(* test hex_to_dword *)
good := good AND HEX_TO_DWORD('0ff') = 255;
good := good AND HEX_TO_DWORD('00') = 0;
good := good AND HEX_TO_DWORD('1') = 1;
good := good AND HEX_TO_DWORD('0A') = 10;
good := good AND HEX_TO_DWORD('0F') = 15;
good := good AND HEX_TO_DWORD('0a') = 10;
good := good AND HEX_TO_DWORD('0f') = 15;
good := good AND HEX_TO_DWORD('00009') = 9;

(* test lowercase *)
good := good AND LOWERCASE('FGTHZuz2345KJGH') = 'fgthzuz2345kjgh';

(* test mirror *)
good := good AND MIRROR('123456789 abc') = 'cba 987654321';

(* test real_to_strf *)
good := good AND REAL_TO_STRF(pi1,2) = '3.14';
good := good AND REAL_TO_STRF(0.015,2) = '0.02';
good := good AND REAL_TO_STRF(0.015,4) = '0.0150';
good := good AND REAL_TO_STRF(0.015,0) = '0';
good := good AND REAL_TO_STRF(3.015,1) = '3.0';
good := good AND REAL_TO_STRF(1234.49967,0) = '1234';
good := good AND REAL_TO_STRF(1234.49967,1) = '1234.5';
good := good AND REAL_TO_STRF(1234.49967,2) = '1234.50';
good := good AND REAL_TO_STRF(1234.49964,3) = '1234.500';
good := good AND REAL_TO_STRF(14.49967,4) = '14.4997';
good := good AND REAL_TO_STRF(1.49967,5) = '1.49967';
good := good AND REAL_TO_STRF(1.49967,6) = '1.499670';

(* test replace_all *)
good := good AND REPLACE_ALL('ab12cd12ef12gh','12','') = 'abcdefgh';
good := good AND REPLACE_ALL('ab12cd12ef12gh','12','21') = 'ab21cd21ef21gh';
good := good AND REPLACE_ALL('ab12cd12ef12gh','12','12') = 'ab12cd12ef12gh';

(* test trim *)
good := good AND TRIM(' ab  cd ef  gh ') = 'abcdefgh';


(* test trim1 *)
good := good AND TRIM1(' ab  cd ef  gh ') = 'ab cd ef gh';

(* test uppercase *)
good := good AND UPPERCASE('fgTHZu z2345KJGH') = 'FGTHZU Z2345KJGH';

(* test capitalize *)
good := good AND CAPITALIZE('hugo wallenstein 123') = 'Hugo Wallenstein 123';

(* test to_upper and to lower *)
FOR t := 0 TO 255 DO
	i := INT_TO_BYTE(t);
	CASE i OF
	0..64:
		good := good AND TO_LOWER(i) = i AND TO_UPPER(i) = i;
	65..90: (* uppercase letters *)
		good := good AND TO_UPPER(i) = i;
		good := good AND TO_LOWER(i) = i + 32;
	91..96:
		good := good AND TO_LOWER(i) = i AND TO_UPPER(i) = i;
	97..122: (* small letters *)
		good := good AND TO_UPPER(i) = i - 32;
		good := good AND TO_LOWER(i) = i;
	123..191:
		good := good AND TO_LOWER(i) = i AND TO_UPPER(i) = i;
	192..214: (* extended uppercase letters *)
		good := good AND TO_UPPER(i) = i;
		good := good AND TO_LOWER(i) = i + 32;
	215:
		good := good AND TO_LOWER(i) = i AND TO_UPPER(i) = i;
	216..222: (* extended uppercase letters *)
		good := good AND TO_UPPER(i) = i;
		good := good AND TO_LOWER(i) = i + 32;
	223:
		good := good AND TO_LOWER(i) = i AND TO_UPPER(i) = i;
	224..246: (* extended lowercase letters *)
		good := good AND TO_UPPER(i) = i-32;
		good := good AND TO_LOWER(i) = i;
	247:
		good := good AND TO_LOWER(i) = i AND TO_UPPER(i) = i;
	248..254: (* extended lowercase letters *)
		good := good AND TO_UPPER(i) = i-32;
		good := good AND TO_LOWER(i) = i;
	255:
		good := good AND TO_LOWER(i) = i AND TO_UPPER(i) = i;
	END_CASE;
	temp := CONCAT(INT_TO_STRING(t),' > ');
	temp := CONCAT(temp,CHR(TO_UPPER(i)));
	temp := CONCAT(temp,' > ');
	temp := CONCAT(temp,CHR(TO_LOWER(i)));
END_FOR;

(* test isc funktionen *)
FOR t := 0 TO 255 DO
	i := INT_TO_BYTE(t);
	CASE i OF
	0..31:
		good := good AND ISC_CTRL(i) = TRUE;
		good := good AND ISC_NUM(i) = FALSE;
		good := good AND ISC_ALPHA(i) = FALSE;
		good := good AND ISC_HEX(i) = FALSE;
		good := good AND ISC_LOWER(i) = FALSE;
		good := good AND ISC_UPPER(i) = FALSE;
	32..47:
		good := good AND ISC_CTRL(i) = FALSE;
		good := good AND ISC_NUM(i) = FALSE;
		good := good AND ISC_ALPHA(i) = FALSE;
		good := good AND ISC_HEX(i) = FALSE;
		good := good AND ISC_LOWER(i) = FALSE;
		good := good AND ISC_UPPER(i) = FALSE;
	48..57:
		good := good AND ISC_CTRL(i) = FALSE;
		good := good AND ISC_NUM(i) = TRUE;
		good := good AND ISC_ALPHA(i) = FALSE;
		good := good AND ISC_HEX(i) = TRUE;
		good := good AND ISC_LOWER(i) = FALSE;
		good := good AND ISC_UPPER(i) = FALSE;
	58..64:
		good := good AND ISC_CTRL(i) = FALSE;
		good := good AND ISC_NUM(i) = FALSE;
		good := good AND ISC_ALPHA(i) = FALSE;
		good := good AND ISC_HEX(i) = FALSE;
		good := good AND ISC_LOWER(i) = FALSE;
		good := good AND ISC_UPPER(i) = FALSE;
	65..70:
		good := good AND ISC_CTRL(i) = FALSE;
		good := good AND ISC_NUM(i) = FALSE;
		good := good AND ISC_ALPHA(i) = TRUE;
		good := good AND ISC_HEX(i) = TRUE;
		good := good AND ISC_LOWER(i) = FALSE;
		good := good AND ISC_UPPER(i) = TRUE;
	75..90:
		good := good AND ISC_CTRL(i) = FALSE;
		good := good AND ISC_NUM(i) = FALSE;
		good := good AND ISC_ALPHA(i) = TRUE;
		good := good AND ISC_HEX(i) = FALSE;
		good := good AND ISC_LOWER(i) = FALSE;
		good := good AND ISC_UPPER(i) = TRUE;
	91..96:
		good := good AND ISC_CTRL(i) = FALSE;
		good := good AND ISC_NUM(i) = FALSE;
		good := good AND ISC_ALPHA(i) = FALSE;
		good := good AND ISC_HEX(i) = FALSE;
		good := good AND ISC_LOWER(i) = FALSE;
		good := good AND ISC_UPPER(i) = FALSE;
	97..102:
		good := good AND ISC_CTRL(i) = FALSE;
		good := good AND ISC_NUM(i) = FALSE;
		good := good AND ISC_ALPHA(i) = TRUE;
		good := good AND ISC_HEX(i) = TRUE;
		good := good AND ISC_LOWER(i) = TRUE;
		good := good AND ISC_UPPER(i) = FALSE;
	103..122:
		good := good AND ISC_CTRL(i) = FALSE;
		good := good AND ISC_NUM(i) = FALSE;
		good := good AND ISC_ALPHA(i) = TRUE;
		good := good AND ISC_HEX(i) = FALSE;
		good := good AND ISC_LOWER(i) = TRUE;
		good := good AND ISC_UPPER(i) = FALSE;
	123..126:
		good := good AND ISC_CTRL(i) = FALSE;
		good := good AND ISC_NUM(i) = FALSE;
		good := good AND ISC_ALPHA(i) = FALSE;
		good := good AND ISC_HEX(i) = FALSE;
		good := good AND ISC_LOWER(i) = FALSE;
		good := good AND ISC_UPPER(i) = FALSE;
	127:
		good := good AND ISC_CTRL(i) = TRUE;
		good := good AND ISC_NUM(i) = FALSE;
		good := good AND ISC_ALPHA(i) = FALSE;
		good := good AND ISC_HEX(i) = FALSE;
		good := good AND ISC_LOWER(i) = FALSE;
		good := good AND ISC_UPPER(i) = FALSE;
	128..191:
		good := good AND ISC_CTRL(i) = FALSE;
		good := good AND ISC_NUM(i) = FALSE;
		good := good AND ISC_ALPHA(i) = FALSE;
		good := good AND ISC_HEX(i) = FALSE;
		good := good AND ISC_LOWER(i) = FALSE;
		good := good AND ISC_UPPER(i) = FALSE;
	192..214:
		good := good AND ISC_CTRL(i) = FALSE;
		good := good AND ISC_NUM(i) = FALSE;
		good := good AND ISC_ALPHA(i) = EXTENDED_ASCII;
		good := good AND ISC_HEX(i) = FALSE;
		good := good AND ISC_LOWER(i) = FALSE;
		good := good AND ISC_UPPER(i) = EXTENDED_ASCII;
	215:
		good := good AND ISC_CTRL(i) = FALSE;
		good := good AND ISC_NUM(i) = FALSE;
		good := good AND ISC_ALPHA(i) = FALSE;
		good := good AND ISC_HEX(i) = FALSE;
		good := good AND ISC_LOWER(i) = FALSE;
		good := good AND ISC_UPPER(i) = FALSE;
	216..222:
		good := good AND ISC_CTRL(i) = FALSE;
		good := good AND ISC_NUM(i) = FALSE;
		good := good AND ISC_ALPHA(i) = EXTENDED_ASCII;
		good := good AND ISC_HEX(i) = FALSE;
		good := good AND ISC_LOWER(i) = FALSE;
		good := good AND ISC_UPPER(i) = EXTENDED_ASCII;
	223:
		good := good AND ISC_CTRL(i) = FALSE;
		good := good AND ISC_NUM(i) = FALSE;
		good := good AND ISC_ALPHA(i) = TRUE;
		good := good AND ISC_HEX(i) = FALSE;
		good := good AND ISC_LOWER(i) = TRUE;
		good := good AND ISC_UPPER(i) = FALSE;
	224..246:
		good := good AND ISC_CTRL(i) = FALSE;
		good := good AND ISC_NUM(i) = FALSE;
		good := good AND ISC_ALPHA(i) = EXTENDED_ASCII;
		good := good AND ISC_HEX(i) = FALSE;
		good := good AND ISC_LOWER(i) = EXTENDED_ASCII;
		good := good AND ISC_UPPER(i) = FALSE;
	247:
		good := good AND ISC_CTRL(i) = FALSE;
		good := good AND ISC_NUM(i) = FALSE;
		good := good AND ISC_ALPHA(i) = FALSE;
		good := good AND ISC_HEX(i) = FALSE;
		good := good AND ISC_LOWER(i) = FALSE;
		good := good AND ISC_UPPER(i) = FALSE;
	248..254:
		good := good AND ISC_CTRL(i) = FALSE;
		good := good AND ISC_NUM(i) = FALSE;
		good := good AND ISC_ALPHA(i) = EXTENDED_ASCII;
		good := good AND ISC_HEX(i) = FALSE;
		good := good AND ISC_LOWER(i) = EXTENDED_ASCII;
		good := good AND ISC_UPPER(i) = FALSE;
	255:
		good := good AND ISC_CTRL(i) = FALSE;
		good := good AND ISC_NUM(i) = FALSE;
		good := good AND ISC_ALPHA(i) = TRUE;
		good := good AND ISC_HEX(i) = FALSE;
		good := good AND ISC_LOWER(i) = TRUE;
		good := good AND ISC_UPPER(i) = FALSE;
	END_CASE;
END_FOR;

(* code test *)
FOR t := 1 TO 255 DO
	good := good AND CODE(CHR(INT_TO_BYTE(t)),1) = INT_TO_BYTE(t);
END_FOR;
temp := '0123456789';
good := good AND CODE(temp,1) = 48;
good := good AND CODE(temp,0) = 0;
good := good AND CODE(temp,11) = 0;
good := good AND CODE(temp,10) = 57;

(* test is_cc is_ncc*)
good := good AND IS_CC('0123456789','0123456789') = TRUE;
good := good AND IS_CC('0 123456789','0123456789') = FALSE;
good := good AND IS_CC('','+-abcdefgh ') = FALSE;
good := good AND IS_NCC('0123456789','+-abcdefgh ') = TRUE;
good := good AND IS_NCC('+0123456789','+-abcdefgh ') = FALSE;
good := good AND IS_NCC('','+-abcdefgh ') = TRUE;

(* test trime *)
good := good AND TRIME('') = '';
good := good AND TRIME('this one') = 'this one';
good := good AND TRIME('  that one   ') = 'that one';

(* test fill *)
good := good AND FILL(32,3) = '   ';
good := good AND FILL(32,0) = '';

(* test fix *)
good := good AND FIX('that one',3,32,0) = 'tha';
good := good AND FIX('this',7,32,0) = 'this   ';
good := good AND FIX('',3,32,0) = '   ';
good := good AND FIX('that one',0,32,0) = '';
good := good AND FIX('that one',3,32,1) = 'one';
good := good AND FIX('this',7,32,1) = '   this';
good := good AND FIX('',3,32,1) = '   ';
good := good AND FIX('that one',0,32,1) = '';
good := good AND FIX('that one',3,32,2) = 'tha';
good := good AND FIX('this',7,32,2) = ' this  ';
good := good AND FIX('',3,32,2) = '   ';
good := good AND FIX('that one',0,32,2) = '';

(* test charcode and charname *)
FOR i := 0 TO 40 DO
	s1 := CHARNAME(i);
	good := good AND (CHARCODE(s1) = i);
END_FOR
good := good AND (CHARNAME(128) = 'euro');
good := good AND (CHARCODE('euro') = 128);




(* revision history
hm	26. mar. 2008	rev 1.0
	original release

hm	29. mar. 2008	rev 1.1
	added trime, fix and fill

hm	29. mar. 2008	rev 1.2
	changed parameter in test fix for new version of fix
	more test for dword_strH

hm	30. mar. 2008	rev 1.3
	added further test for replace UML with € sign

hm	18. may 2008	rev 1.4
	added tests for charcode and charname

*)
END_FUNCTION_BLOCK

(* POU String/FIND_CHAR, ST *)
FUNCTION FIND_CHAR : INT
VAR_INPUT
	str : STRING(STRING_LENGTH);
	pos : INT;
END_VAR
VAR
	i: INT;
	pt : POINTER TO ARRAY[1..255] OF BYTE;
	stop: INT;
	X: BYTE;
END_VAR

(*
version 1.2	29. mar. 2008
programmer 	hugo
tested by		tobias

find_char searches str and returns the starting position of the first character that is not a control character.
control characters are the ascii character 00 .. 31 and 127

*)
pt := ADR(str);
stop := LEN(str);
FOR i := MAX(pos,1) TO stop DO;
	X := pt^[i];
	IF (extended_ascii AND X > 31 AND X <> 127) OR (NOT extended_ascii AND X > 31 AND X < 127) THEN
		FIND_CHAR := i;
		RETURN;
	END_IF;
END_FOR;
FIND_CHAR := 0;


(* revision history
hm	29. feb 2008	rev 1.0
	original version

hm	26. mar. 2008	rev 1.1
	char will now accept extended ascii

hm	29. mar. 2008	rev 1.2
	changed STRING to STRING(STRING_LENGTH)
*)
END_FUNCTION

(* POU String/IS_ALNUM, ST *)
FUNCTION IS_ALNUM : BOOL
VAR_INPUT
	str : STRING(STRING_LENGTH);
END_VAR
VAR
	L: INT;
	pt : POINTER TO BYTE;
	pos: INT;
END_VAR

(*
version 1.1	29. mar. 2008
programmer 		kurt
tested by		hugo

ISC_ALNUM testet ob in einem string nur Zahlen 0..9 vorkommen.

*)
PT := ADR(str);
L := LEN(str);
FOR pos := 1 TO L DO
	IF NOT (ISC_ALPHA(pt^) OR ISC_NUM(pt^)) THEN
		IS_ALNUM := FALSE;
		RETURN;
	END_IF;
    	PT := PT + 1;
END_FOR;
IS_ALNUM := L > 0;


(* revision history
hm	29. feb 2008	rev 1.0
	original version

hm	29. mar. 2008	rev 1.1
	changed STRING to STRING(STRING_LENGTH)
*)
END_FUNCTION

(* POU String/ISC_ALPHA, ST *)
FUNCTION ISC_ALPHA : BOOL
VAR_INPUT
	IN : BYTE;
END_VAR
VAR
END_VAR

(*
version 1.0	6. mar 2008
programmer 	oscat
tested by		hugo

ISC_ALPHA checks if a character is a..z or A..Z.

*)
IF extended_ascii THEN
	ISC_ALPHA := (in > 64 AND in < 91) OR (in > 191  AND in <> 215 AND in <> 247) OR (in > 96 AND in < 123);
ELSE
	ISC_ALPHA := (IN > 64 AND IN < 91) OR (in > 96 AND in < 123);
END_IF;

(* revision history
hm		6. mar. 2008	rev 1.0
	original version

*)
END_FUNCTION

(* POU String/ISC_NUM, ST *)
FUNCTION ISC_NUM : BOOL
VAR_INPUT
	IN : BYTE;
END_VAR
VAR
END_VAR

(*
version 1.0	6. mar 2008
programmer 	oscat
tested by		hugo

ISC_NUM checks if a character is 0..9.

*)
ISC_NUM := IN > 47 AND IN < 58;

(* revision history
hm		6. mar. 2008	rev 1.0
	original version

*)
END_FUNCTION

(* POU String/CHR, ST *)
FUNCTION CHR : STRING(1)
VAR_INPUT
	C : BYTE;
END_VAR
VAR
	PT : POINTER TO BYTE;
END_VAR

(*
version 1.2	29. mar. 2008
programmer 	hugo
tested by		tobias

CHR creates a character from a byte input and stuffs it in a one character length string.

*)
PT := ADR(CHR);
PT^ := C;
pt := pt + 1;
pt^ := 0;

(* revision history
hm	16 jan 2007		rev 1.0
	original version

hm	4. feb. 2008	rev 1.1
	return string would not be terminated properly

hm	29. mar. 2008	rev 1.2
	changed STRING to STRING(1)
*)
END_FUNCTION

(* POU String/IS_ALPHA, ST *)
FUNCTION IS_ALPHA : BOOL
VAR_INPUT
	str : STRING(STRING_LENGTH);
END_VAR
VAR
	L: INT;
	pt : POINTER TO BYTE;
	pos: INT;
END_VAR

(*
version 1.1	29. mar. 2008
programmer 		kurt
tested by		hugo

IS_ALPHA testet ob in einem string nur Zeichen a-z oder A - Z vorkommen.

*)
PT := ADR(str);
L := LEN(str);
FOR pos := 1 TO L DO
	IF NOT ISC_ALPHA(pt^) THEN
		IS_ALPHA := FALSE;
		RETURN;
	END_IF;
    	PT := PT + 1;
END_FOR;
IS_ALPHA := L > 0;


(* revision history
hm	29. feb 2008	rev 1.0
	original version

hm	29. mar. 2008	rev 1.1
	changed STRING to STRING(STRING_LENGTH)
*)
END_FUNCTION

(* POU String/IS_CTRL, ST *)
FUNCTION IS_CTRL : BOOL
VAR_INPUT
	str : STRING(STRING_LENGTH);
END_VAR
VAR
	L: INT;
	pt : POINTER TO BYTE;
	pos: INT;
END_VAR

(*
version 1.1	29. mar 2008
programmer 		kurt
tested by		hugo

IS_CTRL testet ob in einem string nur Steuerzeichen (Char < 32) vorkommen.

*)
PT := ADR(str);
L := LEN(str);
FOR pos := 1 TO L DO
	IF NOT (ISC_CTRL(pt^)) THEN
		IS_CTRL := FALSE;
		RETURN;
	END_IF;
    	PT := PT + 1;
END_FOR;
IS_CTRL := L > 0;


(* revision history
hm	29. feb. 2008	rev 1.0
	original version

hm	29. mar. 2008	rev 1.1
	changed STRING to STRING(STRING_LENGTH)
*)
END_FUNCTION

(* POU String/ISC_CTRL, ST *)
FUNCTION ISC_CTRL : BOOL
VAR_INPUT
	IN : BYTE;
END_VAR
VAR
END_VAR

(*
version 1.0	6. mar 2008
programmer 	oscat
tested by		hugo

ISC_ALPHA checks if a character is a control character.

*)
ISC_CTRL := IN < 32 OR IN = 127;

(* revision history
hm		6. mar. 2008	rev 1.0
	original version

*)
END_FUNCTION

(* POU String/IS_HEX, ST *)
FUNCTION IS_HEX : BOOL
VAR_INPUT
	str : STRING(STRING_LENGTH);
END_VAR
VAR
	L: INT;
	pt : POINTER TO BYTE;
	pos: INT;
END_VAR

(*
version 1.1	29. mar. 2008
programmer 		kurt
tested by		hugo

IS_HEX testet ob in einem string nur Zahlen 0..9 oder A..F oder a..f  vorkommen.

*)
PT := ADR(str);
L := LEN(str);
FOR pos := 1 TO L DO
	IF NOT (ISC_HEX(pt^)) THEN
		IS_HEX := FALSE;
		RETURN;
	END_IF;
    	PT := PT + 1;
END_FOR;
IS_HEX := L > 0;


(* revision history
hm	29. feb 2008	rev 1.0
	original version

hm	29. mar. 2008	rev 1.1
	changed STRING to STRING(STRING_LENGTH)
*)
END_FUNCTION

(* POU String/ISC_HEX, ST *)
FUNCTION ISC_HEX : BOOL
VAR_INPUT
	IN : BYTE;
END_VAR
VAR
END_VAR

(*
version 1.0	6. mar 2008
programmer 	oscat
tested by		hugo

ISC_HEX checks if a character is 0..9, A..F, a..f.

*)
ISC_HEX := (IN > 47 AND IN < 58) OR (IN > 64 AND IN < 71) OR (IN > 96 AND IN < 103);

(* revision history
hm		6. mar. 2008	rev 1.0
	original version

*)
END_FUNCTION

(* POU String/IS_LOWER, ST *)
FUNCTION IS_LOWER : BOOL
VAR_INPUT
	str : STRING(STRING_LENGTH);
END_VAR
VAR
	l: INT;
	pt : POINTER TO BYTE;
	pos: INT;
END_VAR

(*
version 1.1	29. mar. 2008
programmer 		kurt
tested by		hugo

IS_LOWER testet ob in einem string nur kleinbuchstaben vorkommen.

*)
PT := ADR(str);
L := LEN(str);
FOR pos := 1 TO L DO
	IF NOT (ISC_LOWER(pt^)) THEN
		IS_LOWER := FALSE;
		RETURN;
	END_IF;
    	PT := PT + 1;
END_FOR;
IS_LOWER := L > 0;


(* revision history
hm	29. feb 2008	rev 1.0
	original version

hm	29. mar. 2008	rev 1.1
	changed STRING to STRING(STRING_LENGTH)
*)
END_FUNCTION

(* POU String/ISC_LOWER, ST *)
FUNCTION ISC_LOWER : BOOL
VAR_INPUT
	IN : BYTE;
END_VAR
VAR
END_VAR

(*
version 1.0	6 mar 2008
programmer 	hugo
tested by		tobias

isc_lower checks if a character is lowercase.

*)
IF extended_ascii THEN
	ISC_LOWER := ((in > 96) AND (in < 123)) OR ((in > 222) AND (in <> 247));
ELSE
	ISC_LOWER := ((in > 96) AND (in < 123));
END_IF;

(* revision history
hm		6. mar 2008	rev 1.0
	original version

*)
END_FUNCTION

(* POU String/IS_UPPER, ST *)
FUNCTION IS_UPPER : BOOL
VAR_INPUT
	str : STRING(STRING_LENGTH);
END_VAR
VAR
	L: INT;
	pt : POINTER TO BYTE;
	pos: INT;
END_VAR

(*
version 1.1	29. mar. 2008
programmer 		kurt
tested by		hugo

IS_UPPER testet ob in einem string keine Kleinbuchstaben vorkommen.

*)
PT := ADR(str);
L := LEN(str);
FOR pos := 1 TO L DO
	IF NOT (ISC_UPPER(pt^)) THEN
		IS_UPPER := FALSE;
		RETURN;
	END_IF;
    	PT := PT + 1;
END_FOR;
IS_UPPER := L > 0;


(* revision history
hm	29. feb 2008	rev 1.0
	original version

hm	29. mar. 2008	rev 1.1
	changed STRING to STRING(STRING_LENGTH)
*)
END_FUNCTION

(* POU String/ISC_UPPER, ST *)
FUNCTION ISC_UPPER : BOOL
VAR_INPUT
	IN : BYTE;
END_VAR
VAR
END_VAR

(*
version 1.0	6 mar 2008
programmer 	hugo
tested by		tobias

ISC_upper checks if a character is uppercase

*)
IF extended_ascii THEN
	ISC_UPPER :=  ((in > 64) AND (in < 91)) OR (((in > 191) AND (in < 223)) AND (in <> 215));
ELSE
	ISC_UPPER := ((in > 64) AND (in < 91));
END_IF;


(* revision history
hm		6. mar 2008	rev 1.0
	original version

*)
END_FUNCTION

(* POU String/IS_NUM, ST *)
FUNCTION IS_NUM : BOOL
VAR_INPUT
	str : STRING(STRING_LENGTH);
END_VAR
VAR
	L : INT;
	pt : POINTER TO BYTE;
	pos: INT;
END_VAR

(*
version 1.1	29. mar. 2008
programmer 		kurt
tested by		hugo

IS_NUM testet ob in einem string nur Zahlen 0..9 vorkommen.

*)
PT := ADR(str);
L := LEN(str);
FOR pos := 1 TO L DO
	IF NOT (ISC_NUM(pt^)) THEN
		IS_NUM := FALSE;
		RETURN;
	END_IF;
    	PT := PT + 1;
END_FOR;
IS_NUM := L > 0;


(* revision history
hm	29. feb 2008	rev 1.0
	original version

hm	29. mar. 2008	rev 1.1
	changed STRING to STRING(STRING_LENGTH)
*)
END_FUNCTION

(* POU String/REPLACE_UML, ST *)
FUNCTION REPLACE_UML : STRING(STRING_LENGTH)
VAR_INPUT
	str : STRING(STRING_LENGTH);
END_VAR
VAR
	L : INT;
	pt : POINTER TO BYTE;
	pto : POINTER TO BYTE;
	ptm : POINTER TO BYTE;
	pt1, pt2 : POINTER TO BYTE;
	su : STRING(2);
	pos : INT;
END_VAR

(*
version 1.1	29. mar. 2008
programmer 		kurt
tested by		hugo

REPLACE_UML replaces all occurences of Ä,Ö,Ü and ä,ö,ü,ß with Ae, ae, Oe, oe, Ue, ue and ss.

*)
PT := ADR(str);
pto := ADR(REPLACE_UML);
ptm := pto + INT_TO_DWORD(string_length);
pt1 := ADR(su);
pt2 := pt1 + 1;
L := LEN(str);
WHILE pos < L AND pos < string_length DO
	IF pt^ < 127 THEN
		(* no uml character simlply copy the character*)
		pto^ := pt^;
	ELSE
		(* convert the uml character *)
		su := TO_UML(pt^);
		(* we must make sure pointer are not out of range *)
		pto^ := pt1^;
		IF pto < ptm AND pt2^ > 0 THEN
			pto := pto + 1;
			pto^ := pt2^;
		END_IF;
	END_IF;
	(* increment pointers *)
	pt := pt + 1;
	pto := pto + 1;
	pos := pos + 1;
END_WHILE;

(* properly close the output string *)
pto^ := 0;


(* revision history
hm	29. feb 2008	rev 1.0
	original version

hm	29. mar. 2008	rev 1.1
	changed STRING to STRING(STRING_LENGTH)
	new code to avoid pointer out of range
	use new function to_uml
*)
END_FUNCTION

(* POU String/TO_UML, ST *)
FUNCTION TO_UML : STRING(2)
VAR_INPUT
	IN : BYTE;
END_VAR
VAR
END_VAR

(*
version 1.0	29. mar. 2008
programmer 		hugo
tested by		tobias

to_uml converts a character above 127 to a two digit character below 127.
the character Ä is converted to Ae

*)
CASE in OF
	196:	(* Ä *)
		TO_UML := 'Ae';
	214:	(* Ö *)
		TO_UML := 'Oe';
	220:	(* Ü *)
		TO_UML := 'Ue';
	223:	(* ß *)
		TO_UML := 'ss';
	228:	(* ä *)
		TO_UML := 'ae';
	246:	(* ö *)
		TO_UML := 'oe';
	252:	(* ü *)
		TO_UML := 'ue';
ELSE
	TO_UML := CHR(IN);
END_CASE;



(* revision history
hm	29. mar. 2008	rev 1.0
	original version

*)
END_FUNCTION

(* POU String/BYTE_TO_STRH, ST *)
FUNCTION BYTE_TO_STRH : STRING(2)
VAR_INPUT
	IN : BYTE;
END_VAR
VAR
	temp : BYTE;
	PT : POINTER TO BYTE;
END_VAR

(*
version 1.3	29 mar. 2008
programmer 	hugo
tested by		tobias

BYTE_TO_STRINGH converts a Byte to a String of Hexadecimal represented by '0' .. '9' and 'A' .. 'F'.
The lowest order Character will be on the right and the high order Character on the left.

*)
(* read pointer to output string *)
PT := ADR(BYTE_TO_STRH);
(* calculate high order hex value *)
temp := SHR(in,4);
(* convert value to hex character *)
IF temp <= 9 THEN temp := temp + 48; ELSE temp := temp + 55; END_IF;
(* write friat character to output string *)
PT^ := temp;
(* calculate low order hex value *)
temp := in AND 2#00001111;
IF temp <= 9 THEN temp := temp + 48; ELSE temp := temp + 55; END_IF;
(* increment pointer and wirte low order character *)
pt := pt + 1;
pt^ := temp;
(* set pointer at the end of the output string and close the string with 0 *)
pt := pt + 1;
pt^:= 0;


(* code before rev 1.2
FOR i := 1 TO 2 DO
	X := in AND 2#1111;
	IF X <= 9 THEN X := X + 48; ELSE X := X + 55; END_IF;
	Cx := CHR(X);
	temp := CONCAT(Cx, temp);
	in := SHR(in,4);
END_FOR;
BYTE_TO_STRH := temp;
*)

(* revision history

hm	9.6.2007		rev 1.0		
	original version 

hm	11.9.2007		rev 1.1		
	changed coding for compatibility with twincat, under twincat concat cannot have a function as argument.	

hm	15 dec 2007		REV 1.2
	changed code for higher performance

hm	29. mar. 2008	rev 1.3
	changed STRING to STRING(2)
*)
END_FUNCTION

(* POU String/DWORD_TO_STRF, ST *)
FUNCTION DWORD_TO_STRF : STRING(20)
VAR_INPUT
	IN : DWORD;
	N : INT;
END_VAR
VAR
END_VAR

(*
version 1.0	26 jan 2007
programmer 	hugo
tested by		tobias

dword_to_strF converts a DWORD, BYTE or Word to a fixed length String.
the string will be filled with leading zeroes to achieve the fixed length, or if too long, the lowest digits will be used.
the maximum allowed length is 20 mdigits.

for example:	dword_to_strf(123,4) = '0123' 
				dword_to_strf(123,2) = '23'
*)
(* limit N to max 20 characters *)
(* convert dword to string first and cut to length N *)
DWORD_TO_STRF := FIX(DWORD_TO_STRING(in),LIMIT(0,N,20),48,1);


(* revision history
hm	26. jan.2007	rev 1.0		
	original version

hm	29. mar. 2008	rev 1.1
	changed STRING to STRING(20)
	limit the output string to max 20 digits
*)
END_FUNCTION

(* POU String/FIX, ST *)
FUNCTION FIX : STRING(STRING_LENGTH)
VAR_INPUT
	str : STRING(STRING_LENGTH);
	L : INT;
	C : BYTE;
	M : INT;
END_VAR
VAR
	N : INT;
	SX: STRING(STRING_LENGTH);
END_VAR

(*
version 1.0	29. mar. 2008
programmer 	hugo
tested by	tobias

the function fix truncates a string at length L 
or if the string is shorter then L it will be filled with ending Spaces till its length = N.

*)
(* make sure L does not exceed the limits of a string *)
N := LIMIT(0,L,STRING_LENGTH) - LEN(str);
IF N <= 0 THEN
	(* truncate the string at length N *)
	IF M = 1 THEN
		FIX := RIGHT(str,L);
	ELSE
		FIX := LEFT(str,L);
	END_IF;
ELSIF M = 1 THEN
	(* connect fill characters at the beginning *)
	sx := FILL(C,N);
	FIX := CONCAT(sx,str);
ELSIF M = 2 THEN
	(* center str beween fill characters *)
	(* for an uneven number of fill characters, there is one more at the end *)
	sx := FILL(C,SHR(N+1,1));
	FIX := CONCAT(str,sx);
	SX := LEFT(sx,SHR(N,1));
	FIX := CONCAT(sx,FIX);
ELSE
	(* connect fill characters at the end *)
	SX := FILL(C,N);
	FIX := CONCAT(str,SX);
END_IF;


(* revision histroy
hm	29. mar. 2008	rev 1.0
	original release

*)
END_FUNCTION

(* POU String/FILL, ST *)
FUNCTION FILL : STRING(STRING_LENGTH)
VAR_INPUT
	C : BYTE;
	L : INT;
END_VAR
VAR
	i: INT;
	sx: STRING(1);
END_VAR

(*
version 1.0	29. mar. 2008
programmer 	hugo
tested by		tobias

the function fill creates a string at length L of characters C.

*)
Sx := CHR(c);
(* limit L to maximum 80 characters the length of a standard string *)
L := LIMIT(0,L,STRING_LENGTH);
(* create a string of characters to be connected to str *)
FOR i := 1 TO 8 DO
	FILL := CONCAT(FILL,FILL);
	IF L.7 THEN FILL := CONCAT(FILL,Sx); END_IF;
	L := SHL(L,1);
END_FOR;




(* revision histroy
hm	29. mar. 2008	rev 1.0
	original release

*)
END_FUNCTION

(* POU String/EXEC, ST *)
FUNCTION EXEC : STRING(STRING_LENGTH)
VAR_INPUT
	str : STRING(STRING_LENGTH);
END_VAR
VAR
	pos: INT;
	R1: REAL;
	R2: REAL;
	operator: STRING(10);
END_VAR

(*
version 1.4	29. mar. 2008
programmer 	hugo
tested by		tobias

exec executes a mathematical term and returns the result as a string
the term can only be a simple term without brackets and only one operator
allowed operastors are: (+, -, *, /, ^, sqrt, sin, cos, tan).

*)
(* extract both numbers and operator *)
EXEC := UPPERCASE(TRIM(str));

pos := FINDB_NONUM(EXEC);
IF pos > 1 THEN R1 := STRING_TO_REAL(LEFT(EXEC,pos-1)); END_IF;
R2 := STRING_TO_REAL(RIGHT(EXEC,LEN(EXEC)-pos));
EXEC := LEFT(EXEC,pos);
pos := FINDB_NUM(EXEC);
operator := RIGHT(EXEC,LEN(EXEC) - pos);
IF operator = '' AND LEN(str) = 0 THEN
	EXEC := '';
	RETURN;
ELSIF operator = '' THEN
	EXEC := str;
	RETURN;
END_IF;
IF operator = '^' THEN
	EXEC := REAL_TO_STRING(EXPT(R1, R2));
ELSIF operator = 'SQRT' THEN
	EXEC := REAL_TO_STRING(SQRT(R2));
ELSIF operator = 'SIN' THEN
	EXEC := REAL_TO_STRING(SIN(r2));
ELSIF operator = 'COS' THEN
	EXEC := REAL_TO_STRING(COS(r2));
ELSIF operator = 'TAN' THEN
	EXEC := REAL_TO_STRING(TAN(R2));
ELSIF operator = '*' THEN
	EXEC := REAL_TO_STRING(R1 * R2);
ELSIF operator = '/' THEN
	IF R2 <> 0 THEN EXEC := REAL_TO_STRING(R1 / R2); ELSE EXEC := 'ERROR'; END_IF;
ELSIF operator = '+' THEN
	EXEC := REAL_TO_STRING(r1 + r2);
ELSIF operator = '-' THEN
	EXEC := REAL_TO_STRING(r1 - r2);
ELSE
	EXEC := 'ERROR';
END_IF;

IF EXEC = 'ERROR' THEN
	RETURN;
(* some systems deliver integer instead of real *)
ELSIF FIND(EXEC,'.') = 0 THEN
	EXEC := CONCAT(EXEC, '.0');
(* some systems deliver n. instead of n.0 ! *)
ELSIF RIGHT(EXEC,1) = '.' THEN
	EXEC := CONCAT(EXEC,'0');
END_IF;


(* revision history

hm 	6.feb 2007		rev 1.1
	cos has to be written in uppercase
	divide by 0 will return an error

hm	5. mar. 2008	rev 1.2
	add a 0 to the string if a '.' is at the end of the string

hm	20. mar. 2008	rev 1.3
	make sure the function always returns a real value in the form of x.y

hm	29. mar. 2008	rev 1.4
	changed STRING to STRING(STRING_LENGTH)
*)
END_FUNCTION

(* POU String/UPPERCASE, ST *)
FUNCTION UPPERCASE : STRING(STRING_LENGTH)
VAR_INPUT
	str : STRING(STRING_LENGTH);
END_VAR
VAR
	PT : POINTER TO BYTE;
	pos: INT;
	l: INT;
END_VAR

(*
version 1.3	29. mar. 2008
programmer 	hugo
tested by	tobias

uppercase returns str while all letters a..z and ä,ö,ü are converted to uppercase

*)
PT := ADR(UPPERCASE);
uppercase := str;
l := LEN(str);
FOR pos := 1 TO l DO
	pt^ := TO_UPPER(pt^);
	PT := PT + 1;
END_FOR;

(* revision histroy
hm	6. oct. 2006	rev 1.0
	original release

hm	4. feb. 2008	rev 1.1
	improved performance
	added Ä,Ö,Ü

hm	6. mar. 2008	rev 1.2
	added support for exteded Ascii

hm	29. mar. 2008	rev 1.3
	changed STRING to STRING(STRING_LENGTH)
*)	
END_FUNCTION

(* POU String/TO_UPPER, ST *)
FUNCTION TO_UPPER : BYTE
VAR_INPUT
	IN : BYTE;
END_VAR
VAR
END_VAR

(*
version 1.0	6 mar 2008
programmer 	hugo
tested by		tobias

to_upper converts a character from lowercase to uppercase

*)
IF extended_ascii THEN
	IF ((in > 96) AND (in < 123)) OR ((in > 223) AND (in <> 247) AND (in <> 255)) THEN
		TO_UPPER := in AND 16#DF;
	ELSE
		TO_UPPER := in;
	END_IF;
ELSE
	IF ((in > 96) AND (in < 123)) THEN
		TO_UPPER := in AND 16#DF;
	ELSE
		TO_UPPER := in;
	END_IF;
END_IF;

(* revision history
hm		6. mar 2008	rev 1.0
	original version

*)
END_FUNCTION

(* POU String/TRIM, ST *)
FUNCTION TRIM : STRING(STRING_LENGTH)
VAR_INPUT
	str : STRING(STRING_LENGTH);
END_VAR
VAR
	pos: INT;
END_VAR

(*
version 1.2	29. mar. 2008
programmer 	hugo
tested by	tobias

the function deletes all blanks within a string.

*)
TRIM := str;
REPEAT
	pos := FIND(trim,' ');
	IF pos > 0 THEN TRIM := REPLACE(TRIM,'',1,pos); END_IF;
UNTIL pos = 0	END_REPEAT;


(* revision histroy
hm	6.10.2006		rev 1.0
	original release

hm	20. mar. 2008	rev 1.1
	avoid to call replace with pos = 0 because some systems will produce an error

hm	29. mar. 2008	rev 1.2
	changed STRING to STRING(STRING_LENGTH)
*)
END_FUNCTION

(* POU String/FINDB_NONUM, ST *)
FUNCTION FINDB_NONUM : INT
VAR_INPUT
	str : STRING(STRING_LENGTH);
END_VAR
VAR
	pos: INT;
	pt : POINTER TO BYTE;
END_VAR

(*
version 1.2	29. mar. 2008
programmer 	hugo
tested by		tobias

findB_noNum searches str backwards and returns the last position which is not a number.
a number is characterized by a letter "0..9" or "."

*)
pt := ADR(str) + LEN(str) - 1;
FOR pos := LEN(str) TO 1 BY -1 DO;
	IF NOT((PT^ > 47 AND PT^ < 58) OR PT^ = 46) THEN
		FINDB_NONUM := pos;
		RETURN;
	END_IF;
	PT := PT - 1;
END_FOR;
FINDB_NONUM := 0;


(* revision history
hm	6. oct 2006		rev 1.0
	original version

hm	29. feb 2008	rev 1.1
	improved performance

hm	29. mar. 2008	rev 1.2
	changed STRING to STRING(STRING_LENGTH)
*)
END_FUNCTION

(* POU String/FINDB_NUM, ST *)
FUNCTION FINDB_NUM : INT
VAR_INPUT
	str : STRING(STRING_LENGTH);
END_VAR
VAR
	pos: INT;
	pt : POINTER TO BYTE;
END_VAR

(*
version 1.2	29. mar. 2008
programmer 	hugo
tested by	tobias

findB_Num searches str backward and returns the last position of a number
a number is characterized by a letter "0..9" or "."

*)
pt := ADR(str) + LEN(str) - 1;
FOR pos := LEN(str) TO 1 BY -1 DO;
	IF (PT^ > 47 AND PT^ < 58) OR PT^ = 46 THEN
		FINDB_NUM := pos;
		RETURN;
	END_IF;
	PT := PT - 1;
END_FOR;
FINDB_NUM := 0;

(* revision history
hm	6. oct 2006		rev 1.0
	original version

hm	29. feb 2008	rev 1.1
	improved performance

hm	29. mar. 2008	rev 1.2
	changed STRING to STRING(STRING_LENGTH)
*)
END_FUNCTION

(* POU String/COUNT_CHAR, ST *)
FUNCTION COUNT_CHAR : INT
VAR_INPUT
	str : STRING(STRING_LENGTH);
	chr : BYTE;
END_VAR
VAR
	l: INT;
	pt : POINTER TO BYTE;
	pos: INT;
END_VAR


(*
version 1.1	29. mar. 2008
programmer 		kurt
tested by		hugo

COUNT_CHAR how often a character CHAR occurs within a string STR.

*)
PT := ADR(str);
l := LEN(str);
COUNT_CHAR := 0;
FOR pos := 1 TO l DO
	IF pt^ = CHR THEN COUNT_CHAR := COUNT_CHAR + 1; END_IF;
    PT := PT + 1;
END_FOR;


(* revision history
hm	29. feb 2008	rev 1.0
	original version

hm	29. mar. 2008	rev 1.1
	changed STRING to STRING(STRING_LENGTH)
*)
END_FUNCTION

(* POU String/FIND_CTRL, ST *)
FUNCTION FIND_CTRL : INT
VAR_INPUT
	str : STRING(STRING_LENGTH);
	pos : INT;
END_VAR
VAR
	i: INT;
	pt : POINTER TO ARRAY[1..255] OF BYTE;
	stop: INT;
	x: BYTE;
END_VAR

(*
version 1.2	29. mar. 2008
programmer 	hugo
tested by		tobias

find_ctrl searches str and returns the starting position of a control character
control characters are the ascii character 00 .. 31 and 127.

*)
pt := ADR(str);
stop := LEN(str);
FOR i := MAX(pos,1) TO stop DO;
	x := PT^[I];
	IF x < 32 OR X = 127 THEN
		FIND_CTRL := i;
		RETURN;
	END_IF;
END_FOR;
FIND_CTRL := 0;


(* revision history
hm	29. feb 2008	rev 1.0
	original version

hm	26. mar. 2008	rev 1.1
	character 127 is now recognized as control

hm	29. mar. 2008	rev 1.2
	changed STRING to STRING(STRING_LENGTH)
*)
END_FUNCTION

(* POU String/FIND_NONUM, ST *)
FUNCTION FIND_NONUM : INT
VAR_INPUT
	str : STRING(STRING_LENGTH);
	pos : INT;
END_VAR
VAR
	i: INT;
	pt : POINTER TO ARRAY[1..255] OF BYTE;
	end: INT;
	X: BYTE;
END_VAR

(*
version 1.2	29. mar 2008
programmer 	hugo
tested by	tobias

find_noNum searches str and returns the first position which is not a number.
a number is characterized by a letter "0..9" or "."

*)
pt := ADR(str);
end := LEN(str);
FOR i := MAX(pos,1) TO end DO;
	X := pt^[i];
	IF NOT((X > 47 AND X < 58) OR X = 46) THEN
		FIND_NONUM := i;
		RETURN;
	END_IF;
END_FOR;
FIND_NONUM := 0;


(* revision history
hm	6. oct. 2006	rev 1.0
	original version

hm	29. feb 2008	rev 1.1
	added input pos to start search at position

hm	29. mar. 2008	rev 1.2
	changed STRING to STRING(STRING_LENGTH)

*)
END_FUNCTION

(* POU String/FIND_NUM, ST *)
FUNCTION FIND_NUM : INT
VAR_INPUT
	str : STRING(STRING_LENGTH);
	pos : INT;
END_VAR
VAR
	i : INT;
	pt : POINTER TO ARRAY[1..255] OF BYTE;
	stop : INT;
	X: BYTE;
END_VAR

(*
version 1.2	29. mar. 2008
programmer 	hugo
tested by		tobias

find_Num searches str and returns the starting position of a number
a number is characterized by a letter "0..9" or "."

*)
pt := ADR(str);
stop := LEN(str);
FOR i := MAX(pos,1) TO stop DO;
	X := pt^[i];
	IF (X > 47 AND X < 58) OR X = 46 THEN
		FIND_NUM := i;
		RETURN;
	END_IF;
END_FOR;
FIND_NUM := 0;


(* revision history
hm	6. oct. 2006	rev 1.0
	original version

hm	29. feb 2008	rev 1.1
	added input pos to start search at position

hm	29. mar. 2008	rev 1.2
	changed STRING to STRING(STRING_LENGTH)

*)
END_FUNCTION

(* POU String/FINDB, ST *)
FUNCTION FINDB : INT
VAR_INPUT
	str1 : STRING(STRING_LENGTH);
	str2 : STRING(STRING_LENGTH);
END_VAR
VAR
	pos: INT;
	length: INT;
END_VAR

(*
version 1.3	29. mar. 2008
programmer 	hugo
tested by		tobias

the function find searches an str1 for the presence of str2 and returns the first position of str1 of the last presence in instring.
the function is similar to find except it searches from the right to left.
 a 0 is returned if the string is not found.

*)
length := LEN(str2);
FOR pos := LEN(str1) - length + 1 TO 1 BY -1 DO
	IF MID(str1,length,pos) = str2 THEN
		FindB := pos;
		RETURN;
	END_IF;
END_FOR;
FindB := 0;

(* revision history
hm	6. oct 2006		rev 1.0
	original version

hm	15 dec 2007		rev 1.1
	changed code for better performance

hm	29. feb 2008	rev 1.2
	added findb := 0 for compatibility reasons

hm	29. mar. 2008	rev 1.3
	changed STRING to STRING(STRING_LENGTH)
*)
END_FUNCTION

(* POU Engineering/conversion/length, ST *)
FUNCTION_BLOCK length
VAR_INPUT
	m : REAL;
	p : REAL;
	in : REAL;
	ft : REAL;
	yd : REAL;
	mile : REAL;
	sm : REAL;
	fm : REAL;
END_VAR
VAR_OUTPUT
	Ym : REAL;
	Yp : REAL;
	Yin : REAL;
	Yft : REAL;
	Yyd : REAL;
	Ymile : REAL;
	Ysm : REAL;
	Yfm : REAL;
END_VAR
VAR
END_VAR

(*
version 1.0	27 mar 2007
programmer 	hugo
tested by		oscat

this function converts different length units
any unused input can simply be left open.
different inputs connected at the same time will be added up.

*)
Ym :=	m
		+ p * 0.000376065
		+ in * 0.0254
		+ ft * 0.3048
		+ yd * 0.9144
		+ mile * 1609.344
		+ sm * 1852
		+ fm * 1.829;
Yp := Ym / 0.000376065;
Yin := Ym / 0.0254;
Yft := Ym / 0.3048;
Yyd := Ym / 0.9144;
Ymile := Ym / 1609.344;
Ysm := Ym / 1852;
Yfm := Ym / 1.829;

(*
Länge Meter m SI-Basiseinheit
Astronomische Einheit* AE 1 AE = 149,597 870 · E9 m
Parsec pc 1 pc = 206265 AE = 30,857 · E15 m
Lichtjahr Lj 1 Lj = 9,460 530 · E15 m = 63240 AE = 0,306 59 pc
Ångström Å 1 Å = E–l0 m
typograph. Punkt p 1 p = 0,376 065 mm • im Druckereigewerbe
inch** in 1 in = 2,54 · E–2 m = 25,4 mm***
foot ft 1 ft = 0,3048 m = 30,48 cm
yard yd 1 yd = 0,9144 m
mile mile 1 mile = 1609,344 m
Internat. Seemeile sm 1 sm = 1852 m
Fathom fm 1 fm = 1,829 m • in der Seeschifffahrt

*)
END_FUNCTION_BLOCK

(* POU String/FINDP, ST *)
FUNCTION FINDP : INT
VAR_INPUT
	str : STRING(STRING_LENGTH);
	src : STRING(STRING_LENGTH);
	pos: INT;
END_VAR
VAR
	i: INT;
	ls: INT;
	lx: INT;
	stp: INT;
END_VAR

(*
version 1.2	29. mar. 2008
programmer 	hugo
tested by	tobias

the function findP searches a string str for the occurence of src beginning at the position pos.

*)
ls := LEN(str);
lx := LEN(src);
IF ls < lx OR lx = 0 THEN RETURN; END_IF;
stp := ls - lx + 1;
FOR i := MAX(pos,1) TO stp DO
	IF MID(str,lx,i) = src THEN
		FINDP := i;
		RETURN;
	END_IF;
END_FOR;
FINDP := 0;

(* revision histroy
hm	4. feb. 2008	rev 1.0
	original release

hm	29. feb 2008	rev 1.1
	ADDED MAX(pos,1) in loop initialization

hm	29. mar. 2008	rev 1.2
	changed STRING to STRING(STRING_LENGTH)
*)	
END_FUNCTION

(* POU String/HEX_TO_DWORD, ST *)
FUNCTION HEX_TO_DWORD : DWORD
VAR_INPUT
	Hex : STRING(8);
END_VAR
VAR
	pt : POINTER TO BYTE;
	i: INT;
	X: BYTE;
END_VAR

(*
version 1.3	29. mar 2008
programmer 	hugo
tested by	tobias

HEX_TO_DWORD converts a Hexadecimal string into a DWORD.

*)
pt := ADR(hex);
FOR I := 1 TO LEN(hex) DO
	(* read the first character and subtract 48 to get value in decimal 0 = 48 *)
	x := pt^;
	(* calculate the value of the digit *)
	IF X > 47 AND x < 58 THEN
		X := X - 48;
	ELSIF X > 64 AND X < 71 THEN
		X := X - 55;
	ELSIF X > 96 AND X < 103 THEN
		X := X - 87;
	END_IF;
	(* add up the output per hex character which is 4 bits wide *)
	HEX_TO_DWORD := SHL(HEX_TO_DWORD,4) + X;
	pt := pt + 1;
END_FOR

(* revision histroy
hm	2.10.2007		rev 1.0
	original release

hm	19.11.2007		rev 1.1
	changed type of function from int to dword

hm 	4. mar 2008		rev 1.2
	added support for a..f and return 0 for invalid string

hm	29. mar. 2008	rev 1.3
	changed STRING to STRING(STRING_LENGTH)
*)	
END_FUNCTION

(* POU String/LOWERCASE, ST *)
FUNCTION LOWERCASE : STRING(STRING_LENGTH)
VAR_INPUT
	str : STRING(STRING_LENGTH);
END_VAR
VAR
	PT : POINTER TO BYTE;
	pos: INT;
	l: INT;
END_VAR

(*
version 1.3	29. mar. 2008
programmer 	hugo
tested by		tobias

lowercase returns str while all letters A..Z and Ä.Ö,Ü are converted to lowercase.

*)
PT := ADR(LOWERCASE);
lowercase := str;
l := LEN(str);
FOR pos := 1 TO l DO
	pt^ := TO_LOWER(pt^);
	PT := PT + 1;
END_FOR;

(* revision histroy
hm	6. oct. 2006	rev 1.0
	original release

hm	4. feb. 2008	rev 1.1
	improved performance
	added Ä.Ö,Ü

hm	6. mar. 2008	rev 1.2
	added support for exteded Ascii

hm	29. mar. 2008	rev 1.3
	changed STRING to STRING(STRING_LENGTH)
*)	
END_FUNCTION

(* POU String/TO_LOWER, ST *)
FUNCTION TO_LOWER : BYTE
VAR_INPUT
	IN : BYTE;
END_VAR
VAR
END_VAR

(*
version 1.0	6 mar 2008
programmer 	hugo
tested by		tobias

to_lower converts a character from uppercase to lowercase

*)
IF extended_ascii THEN
	IF ((in > 64) AND (in < 91)) OR (((in > 191) AND (in < 223)) AND (in <> 215)) THEN
		TO_LOWER := in OR 16#20;
	ELSE
		TO_LOWER := in;
	END_IF;
ELSE
	IF ((in > 64) AND (in < 91)) THEN
		TO_LOWER := in OR 16#20;
	ELSE
		TO_LOWER := in;
	END_IF;
END_IF;


(* revision history
hm		6. mar 2008	rev 1.0
	original version

*)
END_FUNCTION

(* POU String/MIRROR, ST *)
FUNCTION MIRROR : STRING(STRING_LENGTH)
VAR_INPUT
	str : STRING(STRING_LENGTH);
END_VAR
VAR
	pi : POINTER TO ARRAY[1..255] OF BYTE;
	po : POINTER TO BYTE;
	lx: INT;
	i: INT;
END_VAR

(*
version 1.1	29. mar. 2008
programmer 	hugo
tested by	tobias

this function reverses an input string.

*)
pi := ADR(str);
po := ADR(mirror);
lx := LEN(str);
FOR i := lx TO 1 BY - 1 DO
	po^ := pi^[i];
	po := po + 1;
END_FOR;
(* close output string *)
po^:= 0;


(* revision histroy
hm	4. feb. 2008	rev 1.0
	original release

hm	29. mar. 2008	rev 1.1
	changed STRING to STRING(STRING_LENGTH)
*)	
END_FUNCTION

(* POU String/REAL_TO_STRF, ST *)
FUNCTION REAL_TO_STRF : STRING(20)
VAR_INPUT
	IN : REAL;
	N : INT;
END_VAR
VAR
	O: REAL;
END_VAR

(*
version 1.6	4. apr. 2008
programmer 	hugo
tested by	tobias

Real_to_strF converts a Real to a fixed length String.
the string will be filles with zeroes to achieve the fixed length after the dot.


*)
N := LIMIT(0,N,20);
(* round the input to N digits and convert to string *)
O := in * EXP10(N);
REAL_TO_STRF := DINT_TO_STRING(REAL_TO_DINT(O));
IF LEN(REAL_TO_STRF) < N THEN REAL_TO_STRF := FIX(REAL_TO_STRF, N+1, 48, 1); END_IF;
IF N > 0 THEN REAL_TO_STRF := INSERT(REAL_TO_STRF,'.',LEN(REAL_TO_STRF)-N); END_IF;


(* code used for rev 1.2
(* read pointer to output *)
p1 := ADR(REAL_TO_STRF);
p2 := p1;

(* multiply in with 10^N and truncate *)
FOR I := 1 TO N DO
	temp := temp * 10;
END_FOR;
temp := TRUNC(in * temp + 0.5);
(* multiply temp with in to shift n digits to the left *)
REAL_TO_STRF := DWORD_TO_STRING(temp);
(* now take care of the dot at length - Nth position *)
L := LEN(REAL_TO_STRF);
(* we need to add zero's at the end of the string if there are less then N + 1 zeroes *)
(* this for loop is to align the pointer p1 to the end of the string *)
FOR i := 1 TO L DO p1 := p1 + 1; END_FOR;
FOR i := L TO N DO
	p1^ := 48;
	p1 := p1 + 1;
END_FOR;
(* now we create the space for the dot *)
p2 := p1 - 1;
FOR i := 1 TO N DO
	p1^ := p2^;
	p1 := p1 - 1;
	p2 := p2 - 1;
END_FOR;
(* now we add the dot if N > 0 *)
IF N > 0 THEN
	p1^ := 46;
	(* the string needs to be closed with a 0 at the end *)
	FOR i := 1 TO N + 1 DO p1 := p1 + 1; END_FOR;
	p1^ := 0;
END_IF;
*)

(* code before rev 1.2
dw1 := TRUNC(ABS(in));
dw2 := TRUNC(fract(ABS(in))*exp10(N)+0.5);
IF in < 0 THEN
	s1 := CONCAT('-', DWORD_TO_STRING(dw1));
ELSE
	s1 := DWORD_TO_STRING(dw1);
END_IF;
IF N > 0 THEN s1 := CONCAT(s1, '.'); END_IF;
s2 := DWORD_To_STRF(dw2,N);
Real_To_StrF := CONCAT(s1, s2);
*)

(* revision history
hm		26 jan 2007	rev 1.0
	original version

hm	20. nov. 2007	rev 1.1
	when N=0 ther will be no dot at the end of the string.

hm	15. dec. 2007	rev 1.2
	changed code for better performance

hm	4. mar. 2008	rev 1.3
	result is now rounded instead of trunc

hm	20. mar. 2008	rev 1.4
	changed trunc to real_to_dint because trunc was generating wrong values on wago 842

hm	29. mar. 2008	rev 1.5
	changed STRING to STRING(20)

hm	4. apr. 2008	rev 1.6
	added variable O to avoid an error uner CoDeSys SP PLCWinNT V2.4
*)
END_FUNCTION

(* POU String/REPLACE_ALL, ST *)
FUNCTION REPLACE_ALL : STRING(STRING_LENGTH)
VAR_INPUT
	str : STRING(STRING_LENGTH);
	src : STRING(STRING_LENGTH);
	rep : STRING(STRING_LENGTH);
END_VAR
VAR
	pos: INT;
	lp : INT;
	lx : INT;
END_VAR

(*
version 1.1	29. mar. 2008
programmer 	hugo
tested by	tobias

the function replace_all replaces all occurences of src in str and replaces them by rep.

*)
REPLACE_ALL := str;
lx := LEN(src);
lp := LEN(rep);
pos := FINDP(REPLACE_ALL, src, 1);
WHILE pos > 0 DO
	REPLACE_ALL := REPLACE(REPLACE_ALL,rep,lx, pos);
	pos := FINDP(REPLACE_ALL, src, pos + lp);
END_WHILE;

(* revision histroy
hm	4. feb. 2008	rev 1.0
	original release

hm	29. mar. 2008	rev 1.1
	changed STRING to STRING(STRING_LENGTH)
*)	
END_FUNCTION

(* POU String/TRIM1, ST *)
FUNCTION TRIM1 : STRING(STRING_LENGTH)
VAR_INPUT
	str : STRING(STRING_LENGTH);
END_VAR
VAR
	pos: INT;
END_VAR

(*
version 1.2	29. mar. 2008
programmer 	hugo
tested by		tobias

the function replaces all multiple blanks within a string by only one blank.
leading and ending blanks will be deleted

*)
TRIM1 := str;
REPEAT
	pos := FIND(trim1,'  ');
	IF pos > 0 THEN TRIM1 := REPLACE(TRIM1,' ',2,pos); END_IF;
UNTIL pos = 0	END_REPEAT;
(* beginning and ending blanks need to be stripped off *)
IF LEFT(trim1,1) = ' ' THEN trim1 := DELETE(trim1,1,1); END_IF;
IF RIGHT(trim1,1) = ' ' THEN trim1 := DELETE(trim1,1,LEN(trim1)); END_IF;


(* revision histroy
hm	4. feb. 2008    rev 1.0
	original release

hm	20. mar. 2008	rev 1.1
	avoid to call replace with pos = 0 because some systems will produce an error

hm	29. mar. 2008	rev 1.2
	changed STRING to STRING(STRING_LENGTH)
*)
END_FUNCTION

(* POU String/CAPITALIZE, ST *)
FUNCTION CAPITALIZE : STRING(STRING_LENGTH)
VAR_INPUT
	str : STRING(STRING_LENGTH);
END_VAR
VAR
	PT : POINTER TO BYTE;
	pos : INT;
	L : INT;
	first : BOOL := TRUE;
END_VAR

(*
version 1.1	29. mar 2008
programmer 	hugo
tested by		tobias

uppercase returns str while all letters a..z and ä,ö,ü are converted to uppercase

*)
PT := ADR(CAPITALIZE);
CAPITALIZE := str;
L := LEN(str);
FOR pos := 1 TO l DO
	IF first THEN
		pt^ := TO_UPPER(pt^);
	END_IF;
	(* remember in first if the next char needs to capitalized *)
	IF pt^ = 32 THEN first := TRUE; ELSE first := FALSE; END_IF;
	PT := pt + 1;
END_FOR;

(* revision histroy
hm		4. mar 2008	rev 1.0
	original release

hm	29. mar. 2008	rev 1.1
	changed STRING to STRING(STRING_LENGTH)
*)	
END_FUNCTION

(* POU String/IS_CC, ST *)
FUNCTION IS_CC : BOOL
VAR_INPUT
	str : STRING(STRING_LENGTH);
	cmp : STRING(STRING_LENGTH);
END_VAR
VAR
	L: INT;
	pos: INT;
END_VAR

(*
version 1.1	29. mar. 2008
programmer 	Tobias
tested by	hugo

ISC_CC testet ob ein string nur aus Zeichen des Strings CMP besteht.

*)
L := LEN(str);
FOR pos := 1 TO L DO
	IF FIND(CMP,MID(str,1,pos)) = 0 THEN RETURN; END_IF;
END_FOR;
IS_CC := L > 0;



(* revision history
hm	19. mar 2008	rev 1.0
	original version

hm	29. mar. 2008	rev 1.1
	changed STRING to STRING(STRING_LENGTH)
*)
END_FUNCTION

(* POU String/IS_NCC, ST *)
FUNCTION IS_NCC : BOOL
VAR_INPUT
	str : STRING(STRING_LENGTH);
	cmp : STRING(STRING_LENGTH);
END_VAR
VAR
	L: INT;
	pos: INT;
END_VAR

(*
version 1.1	29. mar. 2008
programmer 		Tobias
tested by		hugo

ISC_NCC testet ob in einem string keine Zeichen des Strings CMP enthalten sind.

*)
L := LEN(str);
FOR pos := 1 TO L DO
	IF FIND(CMP,MID(str,1,pos)) > 0 THEN RETURN; END_IF
END_FOR;
IS_NCC := TRUE;



(* revision history
hm	19. mar 2008	rev 1.0
	original version

hm	29. mar. 2008	rev 1.1
	changed STRING to STRING(STRING_LENGTH)
*)
END_FUNCTION

(* POU String/TRIME, ST *)
FUNCTION TRIME : STRING(STRING_LENGTH)
VAR_INPUT
	str : STRING(STRING_LENGTH);
END_VAR
VAR
END_VAR

(*
version 1.0	28. mar. 2008
programmer 	hugo
tested by	tobias

this function deletes all leading and ending blanks of a string.

*)
TRIME := str;
(* beginning blanks need to be stripped off *)
WHILE LEFT(TRIME,1) = ' ' DO
	TRIME := DELETE(TRIME,1,1);
END_WHILE;

(* ending blanks need to be stripped off *)
WHILE RIGHT(TRIME,1) = ' ' DO
	TRIME := DELETE(TRIME,1,LEN(TRIME));
END_WHILE;


(* revision histroy
hm	28. mar. 2008	rev 1.0
	original release

*)
END_FUNCTION

(* POU String/CHARNAME, ST *)
FUNCTION CHARNAME : STRING(10)
VAR_INPUT
	C : BYTE;
END_VAR
VAR
	search: STRING;
	pos: INT;
END_VAR

(*
version 1.0		13. may. 2008
programmer 		hugo
tested by			hugo

CHARNAME converts a Character code into its HTML character name
ä is convterted to 'äuml'
€ is converted to 'euro'
the character itself is returned if no name is available for the character

*)
CHARNAME := CHR(C);
(* return empty string if code is 0 *)
IF C = 0 THEN RETURN; END_IF;

(* construct search string from code followed by $ sign, also clear charname string*)
search := CONCAT(CHR(C),'&');
search := CONCAT(';', search);

(* search the 4 strings for ocurence and copy the following 10 chars if found*)
pos := FIND(CHARNAME_1, search);
IF pos > 0 THEN
	CHARNAME := MID(CHARNAME_1, 10, pos + 3);
ELSE
	pos := FIND(CHARNAME_2, search);
	IF pos > 0 THEN
		CHARNAME := MID(CHARNAME_2, 10, pos + 3);
	ELSE;
		pos := FIND(CHARNAME_3, search);
		IF pos > 0 THEN
			CHARNAME := MID(CHARNAME_3, 10, pos + 3);
		ELSE
			pos := FIND(CHARNAME_4, search);
			IF pos > 0 THEN CHARNAME := MID(CHARNAME_4, 10, pos + 3); END_IF;
		END_IF;
	END_IF;
END_IF;

(* search for end of name and truncate *)
IF pos > 0 THEN
	pos := FIND(CHARNAME, ';');
	CHARNAME := LEFT(CHARNAME,pos - 1);
END_IF;


(* revision history
hm		13. may. 2008	rev 1.0
	original version

*)
END_FUNCTION

(* POU String/CHARCODE, ST *)
FUNCTION CHARCODE : BYTE
VAR_INPUT
	STR : STRING(10);
END_VAR
VAR
	found: STRING(1);
	search : STRING(10);
	pos: INT;
END_VAR

(*
version 1.0		13. may. 2008
programmer 		hugo
tested by			hugo

CHARCODE converts a HTML Character NAME INTO ITS code
'äuml' is convterted to ä
'euro' is converted to €

*)
(* return 0 if empty string *)
IF str = '' THEN
	RETURN;
ELSIF STR = '&' THEN
	CHARCODE := 33;
	RETURN;
ELSIF str = ';' THEN
	CHARCODE := 59;
	RETURN;
END_IF;

(* construct search string *)
search := CONCAT('&', str);
search := CONCAT(search, ';');

(* search the 4 strings for ocurence and read preceding code if found*)
pos := FIND(CHARNAME_1, search);
IF pos > 0 THEN
	found := MID(CHARNAME_1, 1, pos - 1);
ELSE
	pos := FIND(CHARNAME_2, search);
	IF pos > 0 THEN
		found := MID(CHARNAME_2, 1, pos - 1);
	ELSE
		pos := FIND(CHARNAME_3, search);
		IF pos > 0 THEN
			found := MID(CHARNAME_3, 1, pos - 1);
		ELSE
			pos := FIND(charname_4, search);
			IF pos > 0 THEN found := MID(CHARNAME_4, 1, pos - 1); END_IF;
		END_IF;
	END_IF;
END_IF;

(* convert to code *)
IF pos > 0 THEN
	CHARCODE := CODE(found, 1);
ELSE
	CHARCODE := CODE(STR, 1);
END_IF;


(* revision history
hm		13. may. 2008	rev 1.0
	original version

*)
END_FUNCTION

(* POU XTEST/Testprojekt/array_test, ST *)
FUNCTION_BLOCK array_test
VAR_INPUT
END_VAR
VAR_OUTPUT
	good : BOOL;
END_VAR
VAR CONSTANT
END_VAR
VAR
	test: STRING;
	ax6 : ARRAY[0..6] OF REAL;
	ax7 : ARRAY[0..7] OF REAL;
	ar6 : ARRAY[0..6] OF REAL := 3,2,4,7,1,6,-2;
	(* ar6 median is  	3.0 *)
	(* ar6 average =  	3.0 *)
	(* ar6 sdv =  		3.05505046330389 *)

	ar7 : ARRAY[0..7] OF REAL := -4,6,11,2,9,1,-30,5;
	(* ar7 median is  3.5 *)
	(* ar7 average =  0.0 *)
	(* ar7 sdv =      13.00549334484690 *)
	init : BOOL;
	i: INT;
	X : REAL;
END_VAR
IF NOT init THEN
	init := TRUE;
ELSIF NOT good THEN
	RETURN;
ELSE
	good := FALSE;
END_IF;


(* test _array_init *)
test := '_array_init';
_ARRAY_INIT(ADR(ax6), SIZEOF(ax6),33);
FOR i := 0 TO 6 DO
	IF ax6[i] <> 33 THEN RETURN; END_IF;
END_FOR;
_ARRAY_INIT(ADR(ax7), SIZEOF(ax7), 33);
FOR i := 0 TO 7 DO
	IF ax7[i] <> 33 THEN RETURN; END_IF;
END_FOR;

(* test _array_sort *)
test := '_array_sort';
ax6 := ar6;
_ARRAY_SORT(ADR(ax6),SIZEOF(ax6));
FOR i := 0 TO 5 DO
	IF ax6[i] > ax6[i+1] THEN RETURN; END_IF;
END_FOR;
ax7 := ar7;
_ARRAY_SORT(ADR(ax7),SIZEOF(ax7));
FOR i := 0 TO 6 DO
	IF ax7[i] > ax7[i+1] THEN RETURN; END_IF;
END_FOR;

(* test _array_median *)
test := '_array_median';
ax6 := ar6;
X := _ARRAY_MEDIAN(ADR(ax6),SIZEOF(ax6));
IF NOT CMP(X,3.0,6) THEN RETURN; END_IF;
ax7 := ar7;
X := _ARRAY_MEDIAN(ADR(ax7), SIZEOF(ax7));
IF NOT CMP(X,3.5,6) THEN RETURN; END_IF;

(* test is_sorted *)
test := 'is_sorted';
IF NOT IS_SORTED(ADR(ax6),SIZEOF(ax6)) THEN RETURN; END_IF;
IF NOT IS_SORTED(ADR(ax7),SIZEOF(ax7)) THEN RETURN; END_IF;


(* test _array_shuffle *)
test := '_array_shuffle';
_ARRAY_SHUFFLE(ADR(ax6),SIZEOF(ax6));
_ARRAY_SHUFFLE(ADR(ax7),SIZEOF(ax7));
(* here we have a problem to test *)
(* there is a very little chance that the array is still sorted after array_shuffle *)
IF IS_SORTED(ADR(ax6),SIZEOF(ax6)) THEN RETURN; END_IF;
IF IS_SORTED(ADR(ax7),SIZEOF(ax7)) THEN RETURN; END_IF;
(* be careful theoretically an array can still be sorted after shuffle but chance is very very low *)

(* test array_avg *)
test := 'array_avg';
X := ARRAY_AVG(ADR(ar6),SIZEOF(ar6));
IF NOT CMP(X,3.0,6) THEN RETURN; END_IF;
X := ARRAY_AVG(ADR(ar7), SIZEOF(ar7));
IF NOT CMP(X,0,6) THEN RETURN; END_IF;

(* test array_gav and _array_abs*)
test := 'array_gav';
ax6 := ar6;
_ARRAY_ABS(ADR(ax6), SIZEOF(ax6));
X := ARRAY_GAV(ADR(ax6),SIZEOF(ax6));
IF NOT CMP(X,2.96530981719390,6) THEN RETURN; END_IF;
ax7 := ar7;
_ARRAY_ABS(ADR(ax7), SIZEOF(ax7));
X := ARRAY_GAV(ADR(ax7), SIZEOF(ax7));
IF NOT CMP(X,5.39039959961291,6) THEN RETURN; END_IF;

(* test array_hav *)
test := 'array_hav';
X := ARRAY_HAV(ADR(ax6),SIZEOF(ax6));
IF NOT CMP(X,2.41975308641975,6) THEN RETURN; END_IF;
X := ARRAY_HAV(ADR(ax7), SIZEOF(ax7));
IF NOT CMP(X,3.40133132918188,6) THEN RETURN; END_IF;

(* test array_max *)
test := 'array_max';
IF ARRAY_MAX(ADR(ar6),SIZEOF(ar6)) <> 7 THEN RETURN; END_IF;
IF ARRAY_MAX(ADR(ar7),SIZEOF(ar7)) <> 11 THEN RETURN; END_IF;

(* test aray_min *)
test := 'array_min';
IF ARRAY_MIN(ADR(ar6),SIZEOF(ar6)) <> -2 THEN RETURN; END_IF;
IF ARRAY_MIN(ADR(ar7),SIZEOF(ar7)) <> -30 THEN RETURN; END_IF;

(* test array_sdv *)
test := 'array_sdv';
X := ARRAY_SDV(ADR(ar6),SIZEOF(ar6));
IF NOT CMP(X, 3.05505046330389,6) THEN RETURN; END_IF;
X := ARRAY_SDV(ADR(ar7),SIZEOF(ar7));
IF NOT CMP(X, 13.00549334484690,6) THEN RETURN; END_IF;

(* test array_spr *)
test := 'array_spr';
X := ARRAY_SPR(ADR(ar6),SIZEOF(ar6));
IF NOT CMP(X, 9,6) THEN RETURN; END_IF;
X := ARRAY_SPR(ADR(ar7),SIZEOF(ar7));
IF NOT CMP(X, 41,6) THEN RETURN; END_IF;

(* test aray_sum *)
test := 'array_sum';
IF ARRAY_SUM(ADR(ar6),SIZEOF(ar6)) <> 21 THEN RETURN; END_IF;
IF ARRAY_SUM(ADR(ar7),SIZEOF(ar7)) <> 0 THEN RETURN; END_IF;

(* array_trend *)
test := 'array_trend';
X := ARRAY_TREND(ADR(ar6),SIZEOF(ar6));
IF NOT CMP(X, -1,6) THEN RETURN; END_IF;
X := ARRAY_TREND(ADR(ar7),SIZEOF(ar7));
IF NOT CMP(X, -7.5,6) THEN RETURN; END_IF;

(* array_var *)
test := 'array_var';
X := ARRAY_VAR(ADR(ar6),SIZEOF(ar6));
IF NOT CMP(X, 9.33333333333333,6) THEN RETURN; END_IF;
X := ARRAY_VAR(ADR(ar7),SIZEOF(ar7));
IF NOT CMP(X, 169.14285714285700, 6) THEN RETURN; END_IF;

(* array_add *)
test := 'array_add';
ax6 := ar6;
_ARRAY_ADD(ADR(ax6),SIZEOF(ax6),1);
IF ARRAY_SUM(ADR(ax6),SIZEOF(ax6)) <> 28 THEN RETURN; END_IF;
ax7 := ar7;
_ARRAY_ADD(ADR(ax7),SIZEOF(ax7),1);
IF ARRAY_SUM(ADR(ax7),SIZEOF(ax7)) <> 8 THEN RETURN; END_IF;

(* array_mul *)
test := 'array_mul';
_ARRAY_MUL(ADR(ax6),SIZEOF(ax6),10);
IF ARRAY_SUM(ADR(ax6),SIZEOF(ax6)) <> 280 THEN RETURN; END_IF;
_ARRAY_MUL(ADR(ax7),SIZEOF(ax7),10);
IF ARRAY_SUM(ADR(ax7),SIZEOF(ax7)) <> 80 THEN RETURN; END_IF;



(* set output true if there are no errors *)
test := 'finished';
good := TRUE;


(* revision history
hm	28. mar. 2008	rev 1.0
	original release

hm	29. mar. 2008	rev 1.1
	added further tests to cover all array routines

hm	2. 4. 2008		rev 1.2
	added new array routines

hm	7. apr. 2008	rev 1.3
	rearranged values for ar7 and array trend
*)
END_FUNCTION_BLOCK

(* POU Mathematical/Array/_ARRAY_INIT, ST *)
FUNCTION _ARRAY_INIT : BOOL
VAR_INPUT
	pt : POINTER TO ARRAY[0..32000] OF REAL;
	size : UINT;
	init : REAL;
END_VAR
VAR
	i: UINT;
	stop: UINT;
END_VAR


(*
version 1.3	16 mar 2008
programmer 	hugo
tested by		tobias

this function will initialize a given array with a value init.
the function needs to be called:	_array_init(adr("array"),sizeof("array"));
this function will manipulate a given array.
the function manipulates the original array, it rerturnes true when finished.
because this function works with pointers its very time efficient and it needs no extra memory.

*)
stop := SHR(size,2)-1;
FOR i := 0 TO stop DO
	pt^[i] := init;
END_FOR;

_array_init := TRUE;

(* revision History

hm 6.1.2007		rev 1.1
	change type of function to bool
	added  array_init := true to set output true.

hm	14.11.2007	rev 1.2
	changed stop calculation to be more efficient

hm	16.3. 2008		rev 1.3
	changed type of input size to uint
*)
END_FUNCTION

(* POU Mathematical/Array/_ARRAY_MEDIAN, ST *)
FUNCTION _ARRAY_MEDIAN : REAL
VAR_INPUT
	pt : POINTER TO ARRAY[0..32000] OF REAL;
	size : UINT;
END_VAR
VAR
	i: UINT;
	stop: UINT;
END_VAR

(*
version 1.5	16 mar 2008
programmer 	hugo
tested by		tobias

this function will calculate the median of a given array.
in order to do so the ariginal array is sorted and stays sorted after the function finishes
the function needs to be called:	_array_median(adr("array"),sizeof("array"));
this function will manipulate a given array.
the function will return the median of the original array.
for example [12,0,4,7,1] the median is 4 and the array after the function is called is [0,1,4,7,12]
because this function works with pointers its very time efficient and it needs no extra memory.

*)
_ARRAY_SORT(pt,size);
stop := SHR(size,2)-1;
IF EVEN(UINT_TO_INT(stop)) THEN
	_ARRAY_MEDIAN := pt^[SHR(stop,1)];
ELSE
	i := SHR(stop,1);
	_ARRAY_MEDIAN := (pt^[i] + pt^[i+1]) * 0.5;
END_IF;

(* old code
stop := (size - SIZEOF(pt)) / SIZEOF(pt);
FOR i := 0 TO stop - 1 DO
	FOR m := i + 1 TO stop DO
		IF pt^[i] > pt^[m] THEN
			temp := pt^[i];
			pt^[i] := pt^[m];
			pt^[m] := temp;
		END_IF;
	END_FOR;
END_FOR;
IF even(stop) THEN
	_array_median := pt^[stop/2];
ELSE
	i := stop/2;
	_array_median := (pt^[i] + pt^[i+1])/2;
END_IF;
*)
(* revision history
hm 	3.3.2007		rev 1.1
	corrected an error, changed the statement line 14	i := TRUNC(stop/2); to i := stop/2;

hm		22. sep 2007	rev 1.2
	changed algorithm to use _array_soft for performance reasons

hm		8. oct 2007		rev 1.3
	deleted unused variables m and temp

hm		14. nov 2007	rev 1.4
	corrected a problem with size calculation

hm		16.3. 2008		rev 1.5
	changed type of input size to uint
	performance improvements
*)
END_FUNCTION

(* POU Mathematical/EVEN, ST *)
FUNCTION EVEN : BOOL
VAR_INPUT
	in : DINT;
END_VAR
VAR
END_VAR


(*
version 1.1	1 dec 2007
programmer 	hugo
tested by		tobias

this function chacks an input for even  value
the output is true if the input is even.
execution time on wago 750 - 841 =  10  us
*)
EVEN := NOT in.0;

(* revision history
hm	1. oct 2006	rev 1.0
	ORIGINAL VERSION

hm	01.12.2007	rev 1.1
	changed code for improved performance

hm	21. mar. 2008	rev 1.2
	changed type of input IN from INT to DINT
*)
END_FUNCTION

(* POU Mathematical/Array/IS_SORTED, ST *)
FUNCTION IS_SORTED : BOOL
VAR_INPUT
	pt : POINTER TO ARRAY[0..32000] OF REAL;
	size : UINT;
END_VAR
VAR

	stop: INT;
	i: INT;
END_VAR

(*
version 1.1	4. apr. 2008
programmer 	hugo
tested by	tobias

this function will return true if the given array is sorted in an ascending order.
the function needs to be called:	array_sorted(adr("array"),sizeof("array"));
because this function works with pointers its very time efficient and it needs no extra memory.

*)
stop := UINT_TO_INT(SHR(size,2)-2);
FOR i := 0 TO stop DO
	IF pt^[i] > pt^[i+1] THEN
		IS_SORTED := FALSE;
		RETURN;
	END_IF;
END_FOR;

IS_SORTED := TRUE;

(* revision history

hm 	29. mar. 2008 	rev 1.0
	original version

hm	4. apr. 2008	rev 1.1
	added type conversion to avoid warnings under codesys 3.0
*)
END_FUNCTION

(* POU Mathematical/Array/_ARRAY_SHUFFLE, ST *)
FUNCTION _ARRAY_SHUFFLE : BOOL
VAR_INPUT
	pt : POINTER TO ARRAY[0..32000] OF REAL;
	size : UINT;
END_VAR
VAR
	temp : REAL;
	pos  : INT;
	i: INT;
	stop: INT;
END_VAR


(*
version 1.2	30. mar. 2008
programmer 	kurt
tested by		hugo

this function will randomly shuffle the elements of an array
*)
stop := UINT_TO_INT(SHR(size,2)-1);
FOR i := 0 TO stop DO
        pos := RDM2(i+pos,0,stop);
        (* swap elements *)
        temp := pt^[i];
        pt^[i] := pt^[pos];
        pt^[pos] := temp;
END_FOR;

_ARRAY_SHUFFLE := TRUE;


(* revision History
hm 	4. mar 2008	rev 1.0
	original version

hm	16. mar. 2008	rev 1.1
	changed type of input size to uint

hm	30. mar. 2008	rev 1.2
	changed last in rdm2 fromm pos to i + pos to allow for more randomness

*)
END_FUNCTION

(* POU Mathematical/RDM2, ST *)
FUNCTION RDM2 : INT
VAR_INPUT
	last : INT;
	low : INT;
	high : INT;
END_VAR
VAR
END_VAR




(*
version 1.0	29. feb 2008
programmer 	hugo
tested by	tobias

this function calculates an integer pseudo random number
the random number will be in the range of low <= rdm2 <= high.

*)
RDM2 := TRUNC(RDM(FRACT(last*pi1)) * (high - low + 1)) + low;

(* revision history
hm		29. feb 2008		rev 1.0
	original version

*)
END_FUNCTION

(* POU Mathematical/Array/ARRAY_AVG, ST *)
FUNCTION ARRAY_AVG : REAL
VAR_INPUT
	pt : POINTER TO ARRAY[0..32000] OF REAL;
	size : UINT;
END_VAR
VAR
	i: UINT;
	stop: UINT;
END_VAR

(*
version 1.2	16. mar. 2008
programmer 	hugo
tested by		tobias

this function will calculate the average of a given array.
the function needs to be called:	array_avg(adr("array"),sizeof("array"));
because this function works with pointers its very time efficient and it needs no extra memory.

*)
stop := SHR(size,2)-1;
array_avg := pt^[0];
FOR i := 1 TO stop DO
	array_avg := array_avg + pt^[i];
END_FOR;
array_avg := array_avg / (stop + 1);


(* revision history
hm	2. oct 2007		rev 1.0
	original version

hm	12. dec 2007	rev 1.1
	chaged code for better performance

hm	16. mar. 2008	rev 1.2
	changed input size to uint
*)
END_FUNCTION

(* POU Mathematical/Array/_ARRAY_ABS, ST *)
FUNCTION _ARRAY_ABS : BOOL
VAR_INPUT
	pt : POINTER TO ARRAY[0..32000] OF REAL;
	size : UINT;
END_VAR
VAR
	i: UINT;
	stop: UINT;
END_VAR

(*
version 1.0	2. apr. 2008
programmer 	hugo
tested by	tobias

this function will calculate the absolute value of each element of the array and stroe the result instead of the element.
Array[i] := ABS(ARRAY[i]).
the function needs to be called:	array_avg(adr("array"),sizeof("array"));
because this function works with pointers its very time efficient and it needs no extra memory.

*)
stop := SHR(size,2)-1;
FOR i := 0 TO stop DO
	PT^[i] := ABS(PT^[i]);
END_FOR;
_ARRAY_ABS := TRUE;


(* revision history
hm	2. apr 2008		rev 1.0
	original version

*)
END_FUNCTION

(* POU Mathematical/Array/ARRAY_GAV, ST *)
FUNCTION ARRAY_GAV : REAL
VAR_INPUT
	pt : POINTER TO ARRAY[0..32000] OF REAL;
	size : UINT;
END_VAR
VAR
	i: UINT;
	stop: UINT;
END_VAR

(*
version 1.0	2. apr. 2008
programmer 	hugo
tested by	tobias

this function will calculate the geometric average of a given array.
the function needs to be called:	array_avg(adr("array"),sizeof("array"));
because this function works with pointers its very time efficient and it needs no extra memory.

*)
stop := SHR(size,2)-1;
ARRAY_GAV := 1;
FOR i := 0 TO stop DO
	IF pt^[i] > 0 THEN
		ARRAY_GAV := ARRAY_GAV * pt^[i];
	ELSE
		ARRAY_GAV := 0;
		RETURN;
	END_IF;
END_FOR;
ARRAY_GAV := SQRTN(ARRAY_GAV,UINT_TO_INT(stop)+1);


(* revision history
hm	2. apr 2008		rev 1.0
	original version

*)
END_FUNCTION

(* POU Mathematical/SQRTN, ST *)
FUNCTION SQRTN : REAL
VAR_INPUT
	X : REAL;
	N : INT;
END_VAR
VAR
END_VAR

(*
version 1.2	11. mar 2008
programmer 	hugo
tested by	tobias

this function calculates the nth root function of X according to the formula sqrtn = x^(1/n).

*)
IF N > 0 THEN
	(*	sqrtn := EXPT(x, 1.0 / INT_TO_REAL(n)); old code in rev 1.0 *)
	SQRTN := EXP(LN(x)/n);
ELSE
	SQRTN := 0;
END_IF;


(* revision history
hm		12 jan 2007	rev 1.0
	original version

hm		2. dec 2007	rev 1.1
	changed code for better performance

hm		11. mar 2008	rev 1.2
	added result 0 for compatibility reasons
*)
END_FUNCTION

(* POU Mathematical/Array/ARRAY_HAV, ST *)
FUNCTION ARRAY_HAV : REAL
VAR_INPUT
	pt : POINTER TO ARRAY[0..32000] OF REAL;
	size : UINT;
END_VAR
VAR
	i: UINT;
	stop: UINT;
END_VAR

(*
version 1.0	2. apr. 2008
programmer 	hugo
tested by	tobias

this function will calculate the harmonic average of a given array.
the function needs to be called:	array_avg(adr("array"),sizeof("array"));
because this function works with pointers its very time efficient and it needs no extra memory.

*)
stop := SHR(size,2)-1;
FOR i := 0 TO stop DO
	IF pt^[i] <> 0 THEN
		ARRAY_HAV := ARRAY_HAV + 1/pt^[i];
	ELSE
		ARRAY_HAV := 0;
		RETURN;
	END_IF;
END_FOR;
ARRAY_HAV := (stop + 1) / ARRAY_HAV;


(* revision history
hm	2. apr 2008		rev 1.0
	original version

*)
END_FUNCTION

(* POU Mathematical/Array/ARRAY_MAX, ST *)
FUNCTION ARRAY_MAX : REAL
VAR_INPUT
	pt : POINTER TO ARRAY[0..32000] OF REAL;
	size : UINT;
END_VAR
VAR
	i: UINT;
	stop: UINT;
END_VAR

(*
version 1.1	16. mar. 2008
programmer 	hugo
tested by		tobias

this function will calculate the max value of a given array.
the function needs to be called:	array_max(adr("array"),sizeof("array"));
because this function works with pointers its very time efficient and it needs no extra memory.

*)
stop := (size -SIZEOF(pt)) / SIZEOF(pt);
array_max := pt^[0];
FOR i := 1 TO stop DO
	IF pt^[i] > array_max THEN array_max := pt^[i]; END_IF;
END_FOR;

(* revision history
hm	2. oct 2006		rev 1.0
	original version

hm	16. mar. 2008	rev 1.1
	changed input size to uint
*)
END_FUNCTION

(* POU Mathematical/Array/ARRAY_MIN, ST *)
FUNCTION ARRAY_MIN : REAL
VAR_INPUT
	pt : POINTER TO ARRAY[0..32000] OF REAL;
	size : UINT;
END_VAR
VAR
	i: UINT;
	stop: UINT;
END_VAR

(*
version 1.1	16. mar. 2008
programmer 	hugo
tested by		tobias

this function will calculate the min value of a given array.
the function needs to be called:	array_min(adr("array"),sizeof("array"));
because this function works with pointers its very time efficient and it needs no extra memory.

*)
stop := (size - SIZEOF(pt)) / SIZEOF(pt);
array_min := pt^[0];
FOR i := 1 TO stop DO
	IF pt^[i] < array_min THEN array_min := pt^[i]; END_IF;
END_FOR;


(* revision history
hm		2. oct. 2006
	original version

hm		16. mar. 2008
	changed type of input size to uint

*)
END_FUNCTION

(* POU Mathematical/Array/ARRAY_SDV, ST *)
FUNCTION ARRAY_SDV : REAL
VAR_INPUT
	pt : POINTER TO ARRAY[0..32000] OF REAL;
	size : UINT;
END_VAR
VAR
END_VAR

(*
version 1.1	16. mar 2008
programmer 	hugo
tested by		tobias

this function will calculate the standard deviation of a given array.
the function needs to be called:	array_sdv(adr("array"),sizeof("array"));
because this function works with pointers its very time efficient and it needs no extra memory.

*)
(* standard deviation is simply the square root of the variance *)

array_sdv := SQRT(array_var(pt, size));

(* revision history
hm 	1.4.2007		rev 1.0
	function created

hm	16. mar. 2008	rev 1.1
	changed type of input size to uint

*)
END_FUNCTION

(* POU Mathematical/Array/ARRAY_VAR, ST *)
FUNCTION ARRAY_VAR : REAL
VAR_INPUT
	pt : POINTER TO ARRAY[0..32000] OF REAL;
	size : UINT;
END_VAR
VAR
	avg : REAL;
	i: UINT;
	stop: UINT;
END_VAR

(*
version 1.2	16. mar. 2008
programmer 	hugo
tested by		tobias

this function will calculate the variance of a given array.
the function needs to be called:	array_var(adr("array"),sizeof("array"));
because this function works with pointers its very time efficient and it needs no extra memory.

*)
(* at first we calualte the arithmetic average of the array *)

stop := SHR(size,2)-1;
avg := pt^[0];
FOR i := 1 TO stop DO
	avg := avg + pt^[i];
END_FOR;
avg := avg / (stop + 1);

(* in a second run we calculate the variance of the array *)

array_var := (pt^[0] - avg) * (pt^[0] - avg);
FOR i := 1 TO stop DO
	array_var := array_var + (pt^[i] - avg) * (pt^[i] - avg);
END_FOR;
array_var := array_var / stop;

(* revision history
hm 	1.4.2007	rev 1.0
	function created

hm	12.12.2007	rev 1.1
	changed code for better performance

hm	16. mar. 2008	rev 1.2
	changed type of input size to uint

*)
END_FUNCTION

(* POU Mathematical/Array/ARRAY_SPR, ST *)
FUNCTION ARRAY_SPR : REAL
VAR_INPUT
	pt : POINTER TO ARRAY[0..32000] OF REAL;
	size : UINT;
END_VAR
VAR
	i: UINT;
	stop: UINT;
	array_max : REAL;
	array_min : REAL;
END_VAR

(*
version 1.1	16. mar. 2008
programmer 	hugo
tested by		tobias

this function will calculate the spread of a given array.
the function needs to be called:	array_spr(adr("array"),sizeof("array"));
for example: spread of [12,0,4,1,7] is 12 - 0 = 12.
because this function works with pointers its very time efficient and it needs no extra memory.

*)
stop := (size -SIZEOF(pt)) / SIZEOF(pt);
array_min := pt^[0];
array_max := pt^[0];
FOR i := 1 TO stop DO
	IF pt^[i] > array_max THEN array_max := pt^[i];
	ELSIF pt^[i] < array_min THEN array_min := pt^[i];
	END_IF;
END_FOR;
array_spr := array_max - array_min;


(* revision history
hm 	2. oct. 2006	rev 1.0
	original version

hm	16. mar. 2008	rev 1.1
	changed type of input size to uint

*)
END_FUNCTION

(* POU Mathematical/Array/ARRAY_SUM, ST *)
FUNCTION ARRAY_SUM : REAL
VAR_INPUT
	pt : POINTER TO ARRAY[0..32000] OF REAL;
	size : UINT;
END_VAR
VAR
	i: UINT;
	stop: UINT;
END_VAR


(*
version 1.1	16. mar. 2008
programmer 	hugo
tested by		tobias

this function will calculate the sum of a given array.
the function needs to be called:	array_sum(adr("array"),sizeof("array"));
because this function works with pointers its very time efficient and it needs no extra memory.

*)
stop := (size -SIZEOF(pt)) / SIZEOF(pt);
array_sum := pt^[0];
FOR i := 1 TO stop DO
	array_sum := array_sum + pt^[i];
END_FOR;

(* revision history
hm 	2. oct. 2006	rev 1.0
	function created

hm	16. mar. 2008	rev 1.1
	changed type of input size to uint

*)
END_FUNCTION

(* POU Mathematical/Array/ARRAY_TREND, ST *)
FUNCTION ARRAY_TREND : REAL
VAR_INPUT
	pt : POINTER TO ARRAY[0..32000] OF REAL;
	size : UINT;
END_VAR
VAR
	i: UINT;
	stop: UINT;
	x: REAL;
	stop2: UINT;
END_VAR

(*
version 1.2	16. mar. 2008
programmer 	hugo
tested by		tobias

this function will calculate the trend of a given array.
trend will calculate the avg of the first half of the array and then the avg of the second half, trend = avg2 - avg1.
for example:  [0,1,4,5,3,4,6,3] = 4 - 2.5 = 1.5
the function needs to be called:	array_trend(adr("array"),sizeof("array"));
because this function works with pointers its very time efficient and it needs no extra memory.

*)
stop := SHR(size,2)-1;
stop2 := SHR(stop,1);
FOR i := 0 TO stop2 DO x := x - pt^[i]; END_FOR;
IF EVEN(UINT_TO_INT(stop)) THEN
	FOR i := stop2 TO stop DO X := X + pt^[i]; END_FOR;
ELSE
	FOR i := stop2 + 1 TO stop DO X := X + pt^[i]; END_FOR;
END_IF;
ARRAY_TREND := x / (stop2 + 1);

(* revision history
hm	2 oct 2007	rev 1.0
	original version

hm	12 dec 2007	rev 1.1
	changed code for better performance

hm	16. mar. 2008	rev 1.2
	changed type of input size to uint

*)
END_FUNCTION

(* POU Mathematical/Array/_ARRAY_ADD, ST *)
FUNCTION _ARRAY_ADD : BOOL
VAR_INPUT
	pt : POINTER TO ARRAY[0..32000] OF REAL;
	size : UINT;
	X : REAL;
END_VAR
VAR
	i: UINT;
	stop: UINT;
END_VAR

(*
version 1.0	2. apr. 2008
programmer 	hugo
tested by	tobias

this function will add an offset X to each element of the array and stroe the result instead of the element.
Array[i] := ARRAY[i] + X.
the function needs to be called:	array_avg(adr("array"),sizeof("array"));
because this function works with pointers its very time efficient and it needs no extra memory.

*)
stop := SHR(size,2)-1;
FOR i := 0 TO stop DO
	PT^[i] := PT^[i] + X;
END_FOR;
_ARRAY_ADD := TRUE;


(* revision history
hm	2. apr 2008		rev 1.0
	original version

*)
END_FUNCTION

(* POU Mathematical/Array/_ARRAY_MUL, ST *)
FUNCTION _ARRAY_MUL : BOOL
VAR_INPUT
	pt : POINTER TO ARRAY[0..32000] OF REAL;
	size : UINT;
	X : REAL;
END_VAR
VAR
	i: UINT;
	stop: UINT;
END_VAR

(*
version 1.0	2. apr. 2008
programmer 	hugo
tested by	tobias

this function will multiply each element of the array and stroe the result instead of the element.
Array[i] := ARRAY[i] * X.
the function needs to be called:	array_avg(adr("array"),sizeof("array"));
because this function works with pointers its very time efficient and it needs no extra memory.

*)
stop := SHR(size,2)-1;
FOR i := 0 TO stop DO
	PT^[i] := PT^[i] * X;
END_FOR;
_ARRAY_MUL := TRUE;


(* revision history
hm	2. apr 2008		rev 1.0
	original version

*)
END_FUNCTION

(* POU XTEST/Testprojekt/DATE_TEST, ST *)
FUNCTION_BLOCK DATE_TEST
VAR_INPUT
END_VAR
VAR_OUTPUT
	good : BOOL;
END_VAR
VAR
	INIT : BOOL;
	rx : DWORD;
	XD: DATE;
	YD : DATE;
	xdt : DT;
	test: STRING;
	rr: REAL;
	s1: STRING;
	yr : INT;
	mth : INT;
	day : INT;
	hr: INT;
	m: INT;
	sec: INT;
	tb: BOOL;
	ti: INT;
	tdt: DT;
	tde: DT;
	te: INT;
	wd : INT;
	wdi : DINT;
	tt: TIME;
END_VAR
IF NOT init THEN
	init := TRUE;
ELSIF NOT good THEN
	RETURN;
ELSE
	good := FALSE;
END_IF;

(* prepare random numbers *)
rx := RDMDW(rx);

(* the maximum defindes date for oscat functions is 2099-12-31-23:59:59 *)
IF rx > 4102444799 THEN rx := rx - 200000000; END_IF;

rr := RDM(rr);
(* generate random date and randon dt *)
xdt := DWORD_TO_DT(rx);

(* analyze date *)
s1 := DT_TO_STRING(xdt);
s1 := RIGHT(s1, LEN(s1)-FIND(s1,'#'));
yr := STRING_TO_INT(LEFT(s1,4));
s1 := RIGHT(s1, LEN(s1)-FIND(s1,'-'));
mth := STRING_TO_INT(LEFT(s1,2));
s1 := RIGHT(s1, LEN(s1)-FIND(s1,'-'));
day := STRING_TO_INT(LEFT(s1,2));
(* analyze Time *)
s1 := RIGHT(s1, LEN(s1)-FIND(s1,'-'));
hr := STRING_TO_INT(LEFT(s1,2));
s1 := RIGHT(s1, LEN(s1)-FIND(s1,':'));
m := STRING_TO_INT(LEFT(s1,2));
s1 := RIGHT(s1, LEN(s1)-FIND(s1,':'));
sec := STRING_TO_INT(LEFT(s1,2));

(*
xd := DT_TO_DATE(xdt);
dt_to Date delivers wrong result when year > 2038
*)
xd := set_Date(yr,mth,day);

(* test set_date *)
test := 'set_date';
IF set_Date(yr,mth,day) <> xd THEN RETURN; END_IF;

(* test set_dt *)
test := 'set_dt';
IF set_DT(yr,mth,day,hr,m,sec) <> xdt THEN RETURN; END_IF;

(* test date_add *)
test := 'date_add';
YD := date_add(xd,0,0,0,0);
IF YD <> XD THEN RETURN; END_IF;
yd := date_add(d#2000-1-1,5,0,0,0);
IF yd <> d#2000-1-6 THEN RETURN; END_IF;
yd := date_add(d#2000-1-1,-31,0,0,0);
IF yd <> d#1999-12-1 THEN RETURN; END_IF;
yd := date_add(d#2000-1-1,60,0,0,0);
IF yd <> d#2000-3-1 THEN RETURN; END_IF;
yd := date_add(d#2001-1-1,59,0,0,0);
IF yd <> d#2001-3-1 THEN RETURN; END_IF;
yd := date_add(d#2002-1-1,59,0,0,0);
IF yd <> d#2002-3-1 THEN RETURN; END_IF;
yd := date_add(d#2003-1-1,59,0,0,0);
IF yd <> d#2003-3-1 THEN RETURN; END_IF;
yd := date_add(d#2004-1-1,60,0,0,0);
IF yd <> d#2004-3-1 THEN RETURN; END_IF;
yd := date_add(d#2000-1-1,0,1,0,0);
IF yd <> d#2000-1-8 THEN RETURN; END_IF;
yd := date_add(d#2000-1-1,0,-1,0,0);
IF yd <> d#1999-12-25 THEN RETURN; END_IF;
yd := date_add(d#2000-1-1,0,0,12,0);
IF yd <> d#2001-1-1 THEN RETURN; END_IF;
yd := date_add(d#2000-1-1,0,0,-1,0);
IF yd <> d#1999-12-1 THEN RETURN; END_IF;
yd := date_add(d#2000-1-1,0,0,0,99);
IF yd <> d#2099-1-1 THEN RETURN; END_IF;
yd := date_add(d#2000-1-1,0,0,0,-12);
IF yd <> d#1988-1-1 THEN RETURN; END_IF;
yd := date_add(d#2000-1-1,-31,1,1,1);
IF yd <> d#2001-1-8 THEN RETURN; END_IF;
yd := date_add(d#2000-1-1,31,1,-1,-1);
IF yd <> d#1999-1-8 THEN RETURN; END_IF;

(* test day_of_date *)
test := 'day_of_date';
IF day_of_date(XD) <> DATE_TO_DWORD(xd) / 86400 THEN RETURN; END_IF;

(* test day_of_month *)
test := 'day_of_month';
IF day_of_month(xd) <> day THEN RETURN; END_IF;

(* test day_of_year *)
test := 'day_of_year';
IF day_of_date(xd) - day_of_date(set_Date(yr,1,1)) + 1 <> day_of_year(xd) THEN RETURN; END_IF;

(* test days_delta *)
test := 'days_delta';
IF days_delta(xd, xd) <> 0 THEN RETURN; END_IF;
IF days_delta(D#2008-1-1,D#2007-12-31) <> -1 THEN RETURN; END_IF;
IF days_delta(D#2008-2-28,D#2008-3-1) <> 2 THEN RETURN; END_IF;
IF days_delta(D#2012-3-1,D#2012-2-28) <> -2 THEN RETURN; END_IF;
IF days_delta(D#2007-2-28,D#2007-3-1) <> 1 THEN RETURN; END_IF;
IF days_delta(D#1970-1-1,xd) <> day_of_date(xd) THEN RETURN; END_IF;

(* test DST *)
(*
Equation used TO calculate the beginning OF European Summer TIME:
Sunday (31 - (5*y/4 + 4) mod 7) March at 01.00 UTC
(valid through 2099, courtesy of Robert H. van Gent, EC).
European Summer Time ends (clocks go back) at 01.00 UTC on

    * 29 October 2006
    * 28 October 2007
    * 26 October 2008

Equation used to calculate the end of European Summer Time:
Sunday (31 - (5*y/4 + 1) mod 7) October at 01.00 UTC
(validity AND credits as above).
*)
test := 'dst';
ti := 31 -(5*yr/4 + 4) MOD 7;
te := 31-(5*yr/4+1) MOD 7;
tdt := set_DT(yr,3,ti,1,0,0);
tde := set_DT(yr,10,te,1,0,0);
tb := xdt >= tdt AND xdt < tde;
IF DST(xdt) <> tb THEN RETURN; END_IF;
IF DST(tdt) = FALSE THEN RETURN; END_IF;
tdt := set_DT(yr,3,ti,0,59,59);
IF DST(tdt) = TRUE THEN RETURN; END_IF;
tdt := set_DT(yr,10,te,0,59,59);
IF DST(tdt) = FALSE THEN RETURN; END_IF;
IF DST(tde) = TRUE THEN RETURN; END_IF;

(* easter test *)
test := 'easter';
IF easter_test() <> TRUE THEN RETURN; END_IF;

(* test leap_of_date *)
test := 'leap_of_Date';
tb := yr MOD 4 = 0;
IF leap_of_Date(xd) <> tb THEN RETURN; END_IF;

(* test leap_year *)
test := 'leap_year';
IF leap_year(yr) <> tb THEN RETURN; END_IF;

(* test local_time *)
test := 'local_time';
TT := T#12h;
IF local_time(xdt,-12,FALSE) <> xdt - TT THEN RETURN; END_IF;
IF local_time(xdt,0,FALSE) <> xdt THEN RETURN; END_IF;
TT := T#1h;
IF local_time(xdt,1,FALSE) <> xdt + TT THEN RETURN; END_IF;
TT := T#12h;
IF local_time(xdt,+12,FALSE) <> xdt + TT THEN RETURN; END_IF;
IF DST(xdt) THEN
	TT := T#11h;
	IF local_time(xdt,-12,TRUE) <> xdt - TT THEN RETURN; END_IF;
	TT := T#1h;
	IF local_time(xdt,0,TRUE) <> xdt + TT THEN RETURN; END_IF;
	TT := T#2h;
	IF local_time(xdt,1,TRUE) <> xdt + TT THEN RETURN; END_IF;
	TT := T#13h;
	IF local_time(xdt,+12,TRUE) <> xdt + TT THEN RETURN; END_IF;
ELSE
	TT := T#12h;
	IF local_time(xdt,-12,TRUE) <> xdt - TT THEN RETURN; END_IF;
	IF local_time(xdt,0,TRUE) <> xdt THEN RETURN; END_IF;
	TT := T#1h;
	IF local_time(xdt,1,TRUE) <> xdt + TT THEN RETURN; END_IF;
	TT := T#12h;
	IF local_time(xdt,+12,TRUE) <> xdt + TT THEN RETURN; END_IF;
END_IF;

(* ltime_to_utc *)
test := 'ltime_to_utc';
TT := T#1h;
IF Ltime_to_UTC(xdt+TT,FALSE,1) <> xdt THEN RETURN; END_IF;
IF Ltime_to_UTC(xdt - TT, FALSE,-1) <> xdt THEN RETURN; END_IF;
IF Ltime_to_UTC(xdt, FALSE,0) <> xdt THEN RETURN; END_IF;
TT := T#2h;
IF Ltime_to_UTC(xdt+ TT,TRUE,1) <> xdt THEN RETURN; END_IF;
IF Ltime_to_UTC(xdt, TRUE,-1) <> xdt THEN RETURN; END_IF;
TT := T#1h;
IF Ltime_to_UTC(xdt + TT, TRUE,0) <> xdt THEN RETURN; END_IF;

(* month test *)
test := 'month';
IF month(xd) <> mth THEN RETURN; END_IF;

(* period test *)
test := 'period';
yd := set_Date(2000,mth,day);
IF period(d#2000-3-3,xd,d#2000-9-3) <> (yd >= d#2000-3-3 AND yd <= d#2000-9-3) THEN RETURN; END_IF;
IF period(d#2000-9-3,xd,d#2000-3-3) <> (yd <= d#2000-3-3 OR yd >= d#2000-9-3) THEN RETURN; END_IF;

(* test weekday *)
test := 'weekday';
wd := weekday(xd);
wdi := DWORD_TO_DINT(DATE_TO_DWORD(xd)/86400);
wdi := (wdi + 4) MOD 7;
IF wdi = 0 THEN wdi := 7; END_IF;
IF wd <> wdi THEN RETURN; END_IF;

(* test year *)
test := 'year';
IF year(xd) <> yr THEN RETURN; END_IF;

(* test year_begin *)
test := 'year_begin';
IF year_begin(yr) <> set_Date(yr,1,1) THEN RETURN; END_IF;

(* test work_week *)
test := 'work_week';
IF NOT work_week_test() THEN RETURN; END_IF;

(* set output true if there are no errors *)
test := 'finished';
good := TRUE;


(* revision history
hm		26. mar. 2008		rev 1.0
	original release

*)
END_FUNCTION_BLOCK

(* POU Mathematical/RDMDW, ST *)
FUNCTION RDMDW : DWORD
VAR_INPUT
	last : DWORD;
END_VAR
VAR
	RX: REAL;
	M: REAL;
END_VAR




(*
version 1.1	18. may. 2008
programmer 	hugo
tested by		tobias

this function calculates a DWORD pseudo random number.

*)
M := BIT_COUNT(last);
RX := RDM(FRACT(M*pi1));
RDMDW := SHL(REAL_TO_DWORD(rx*65535),16);
RX := RDM(FRACT(M * E1));
RDMDW := RDMDW OR (REAL_TO_DWORD(rx*65535) AND 16#0000FFFF);



(* revision history
hm		14. mar 2008		rev 1.0
	original version

hm		18. may. 2008		rev 1.1
	changed constant E to E1
*)
END_FUNCTION

(* POU Time&Date/SET_DT, ST *)
FUNCTION SET_DT : DT
VAR_INPUT
	year : INT;
	month : INT;
	day : INT;
	hour : INT;
	minute : INT;
	second : INT;
END_VAR
VAR
END_VAR

(*
version 1.5	16 mar 2008
programmer 	hugo
tested by	tobias


creates a date output from year, month and day of month
year must be in the form of 4 digits ie 2006 or 1977.
*)
set_DT := DWORD_TO_DT(DATE_TO_DWORD(set_Date(year, month, day)) + INT_TO_DWORD(second) + INT_TO_DWORD(minute) * 60 + INT_TO_DWORD(hour) * 3600);


(* revision history
hm	4. aug. 2006		rev 1.0
	original version

hm		19 sep. 2007	rev 1.1
	use function leap_year to calculate leap year, more exceptions are handled

hm		1. okt 2007		rev 1.2
	added step7 compatibility
	call function set_date

hm		8. oct 2007		rev 1.3
	deleted unused variables count and leap

hm		1. 11 2007		rev 1.4
	converted hour type integer to dword in calculation to avoid overrun on möller ecp4

hm		16. mar 2008	rev 1.5
	added type conversions to avoid warnings under codesys 3.0
*)
END_FUNCTION

(* POU Time&Date/HOUR, ST *)
FUNCTION HOUR : INT
VAR_INPUT
	itod : TOD;
END_VAR
VAR
END_VAR

(*
version 1.1	2 okt 2006
programmer 	hugo
tested by	tobias

extracts the hour of a Time_of_day 
*)
hour := DWORD_TO_INT(TOD_TO_DWORD(itod)/3600000);


(* change history
hm 4. aug 2006	rev 1.0
	original version

hm 2.10.2006 	rev 1.1
	changed name of input to itod

*)
END_FUNCTION

(* POU Time&Date/MINUTE, ST *)
FUNCTION MINUTE : INT
VAR_INPUT
	itod : TOD;
END_VAR
VAR
END_VAR

(*
version 1.1	2 oct 2006
programmer 	hugo
tested by		tobias

extracts the minutes out of TOD truncating the ceconds 

*)  
minute := DWORD_TO_INT(TOD_TO_DWORD(itod)/60000 - TOD_TO_DWORD(itod)/3600000 * 60);


(* change history

2.10.2006 changes name of input to itod

*)
END_FUNCTION

(* POU Time&Date/SECOND, ST *)
FUNCTION SECOND : REAL
VAR_INPUT
	itod : TOD;
END_VAR
VAR
END_VAR

(*
version 1.1	2 oct 2006
programmer 	hugo
tested by		tobias

returns the seconds and milliseconds as real of TOD   
 
*)
second := DWORD_TO_REAL(TOD_TO_DWORD(itod) - TOD_TO_DWORD(itod)/60000 * 60000)/1000;



(* change history

2.10.2006 changes name of input to itod

*)
END_FUNCTION

(* POU Time&Date/DAY_OF_DATE, ST *)
FUNCTION DAY_OF_DATE : DINT
VAR_INPUT
	idate : DATE;
END_VAR
VAR
END_VAR


(*
	version 1.3	7. apr. 2008
	programmer 	oscat
	tested BY	oscat

DAY_OF_DATE returns the days since 1.1.1970

*)
day_of_date := DWORD_TO_DINT(DATE_TO_DWORD(idate) / 86400);


(* revision history
hm		16.9.2007		rev 1.0
	original version

hm		1. okt 2007		rev 1.1
	added step7 compatibility

hm		22. mar. 2008	rev 1.2
	changed output from int to Dint because the total date range is 49710 days

hm		7. apr. 2008	rev 1.3
	deleted unused step7 code

*)
END_FUNCTION

(* POU Time&Date/DAYS_DELTA, ST *)
FUNCTION DAYS_DELTA : DINT
VAR_INPUT
	date_1 : DATE;
	date_2 : DATE;
END_VAR
VAR
END_VAR

(*
version 1.2	22. mar. 2008
programmer 	hugo
tested by		tobias

days_delta calculates the days between two dates. the days are calculated date_2 - date_1.

*)
days_delta := day_of_date(date_2) - day_of_date(date_1);

(* revision history
hm	27. dec 2006	rev 1.0
	original version

hm	16.9.2007		rev 1.1
	coorected an error in formula and changed algorithm to show positive and negative delta

hm	22. mar. 2008	rev 1.2
	changed output from int to dint because the total date range is 49710 days
*)
END_FUNCTION

(* POU Time&Date/DST, ST *)
FUNCTION DST : BOOL
VAR_INPUT
	utc : DT;
END_VAR
VAR
	yr : INT;
	yr4 : DWORD;
	ltc: DWORD;
	idate : DWORD;
END_VAR

(*
version 1.3	16. mar. 2008
programmer 	hugo
tested by		tobias

this functions returns TRUE IF dst TIME is active 
the FUNCTION calculates automatically for any year betweek 1970 AND 2099 
wheather daylight savings is on OR off 
the summertime calculation is done according to european standards.
dst will become TRUE AT 01:00 utc in the morning FOR the respective days 
AND it will become FALSE after daylight savings TIME is switched back end OF october at 01:00 utc

*)
yr := year(DT_TO_DATE(utc));
ltc := DT_TO_DWORD(utc);
idate := DT_TO_DWORD(set_DT(yr,3,31,1,0,0));
yr4 := SHR(5*INT_TO_DWORD(yr),2);
DST := (idate - ((yr4+4) MOD 7)*86400 <= ltc) AND (idate + (214 - (yr4+1) MOD 7)*86400 > ltc);

(* revision history
hm	4. aug 2006	rev 1.0
	original version

hm	24. okt 2007	rev 1.1
	deleted time_zone_offset input because dst is generally at 01:00 utc and not mesz
	uk starts 01:00 utc and also greece

hm	1. dec 2007	rev 1.2
	changed code to improve performance

hm	16. mar. 2008	rev 1.3
	added type conversion to avoid warnings under codesys 3.0
	code improvement for better performance

*)

(*
Equation used TO calculate the beginning OF European Summer TIME:
Sunday (31 - (5*y/4 + 4) mod 7) March at 01.00 UTC
(valid through 2099, courtesy of Robert H. van Gent, EC).

European Summer Time ends (clocks go back) at 01.00 UTC on

    * 29 October 2006
    * 28 October 2007
    * 26 October 2008

Equation used to calculate the end of European Summer Time:
Sunday (31 - (5*y/4 + 1) mod 7) October at 01.00 UTC
(validity AND credits as above).

*)
END_FUNCTION

(* POU XTEST/Testprojekt/TEST Routines/easter_test, ST *)
FUNCTION easter_test : BOOL
VAR_INPUT
END_VAR
VAR
	x: BOOL := TRUE;
END_VAR
x := easter(1980) = d#1980-4-6;
x := easter(1981) = d#1981-4-19 AND x;
x := easter(1982) = d#1982-4-11 AND x;
x := easter(1983) = d#1983-4-3 AND x;
x := easter(1984) = d#1984-4-22 AND x;
x := easter(1985) = d#1985-4-7 AND x;
x := easter(1986) = d#1986-3-30 AND x;
x := easter(1987) = d#1987-4-19 AND x;
x := easter(1988) = d#1988-4-3 AND x;
x := easter(1989) = d#1989-3-26 AND x;
x := easter(1990) = d#1990-4-15 AND x;
x := easter(1991) = d#1991-3-31 AND x;
x := easter(1992) = d#1992-4-19 AND x;
x := easter(1993) = d#1993-4-11 AND x;
x := easter(1994) = d#1994-4-3 AND x;
x := easter(1995) = d#1995-4-16 AND x;
x := easter(1996) = d#1996-4-7 AND x;
x := easter(1997) = d#1997-3-30 AND x;
x := easter(1998) = d#1998-4-12 AND x;
x := easter(1999) = d#1999-4-4 AND x;
x := easter(2000) = d#2000-4-23 AND x;
x := easter(2001) = d#2001-4-15 AND x;
x := easter(2002) = d#2002-3-31 AND x;
x := easter(2003) = d#2003-4-20 AND x;
x := easter(2004) = d#2004-4-11 AND x;
x := easter(2005) = d#2005-3-27 AND x;
x := easter(2006) = d#2006-4-16 AND x;
x := easter(2007) = d#2007-4-8 AND x;
x := easter(2008) = d#2008-3-23 AND x;
x := easter(2009) = d#2009-4-12 AND x;
x := easter(2010) = d#2010-4-4 AND x;
x := easter(2011) = d#2011-4-24 AND x;
x := easter(2012) = d#2012-4-8 AND x;
x := easter(2013) = d#2013-3-31 AND x;
x := easter(2014) = d#2014-4-20 AND x;
x := easter(2015) = d#2015-4-5 AND x;
x := easter(2016) = d#2016-3-27 AND x;
x := easter(2017) = d#2017-4-16 AND x;
x := easter(2018) = d#2018-4-1 AND x;
x := easter(2019) = d#2019-4-21 AND x;
x := easter(2020) = d#2020-4-12 AND x;
x := easter(2021) = d#2021-4-4 AND x;
x := easter(2022) = d#2022-4-17 AND x;
x := easter(2023) = d#2023-4-9 AND x;
x := easter(2024) = d#2024-3-31 AND x;
x := easter(2025) = d#2025-4-20 AND x;
x := easter(2026) = d#2026-4-5 AND x;
x := easter(2027) = d#2027-3-28 AND x;
x := easter(2028) = d#2028-4-16 AND x;
x := easter(2029) = d#2029-4-1 AND x;
x := easter(2030) = d#2030-4-21 AND x;
x := easter(2031) = d#2031-4-13 AND x;
x := easter(2032) = d#2032-3-28 AND x;
x := easter(2033) = d#2033-4-17 AND x;
x := easter(2034) = d#2034-4-9 AND x;
x := easter(2035) = d#2035-3-25 AND x;
x := easter(2036) = d#2036-4-13 AND x;
x := easter(2037) = d#2037-4-5 AND x;
x := easter(2038) = d#2038-4-25 AND x;
x := easter(2039) = d#2039-4-10 AND x;
x := easter(2040) = d#2040-4-1 AND x;
x := easter(2041) = d#2041-4-21 AND x;
x := easter(2042) = d#2042-4-6 AND x;
x := easter(2043) = d#2043-3-29 AND x;
x := easter(2044) = d#2044-4-17 AND x;
x := easter(2045) = d#2045-4-9 AND x;
x := easter(2046) = d#2046-3-25 AND x;
x := easter(2047) = d#2047-4-14 AND x;
x := easter(2048) = d#2048-4-5 AND x;
x := easter(2049) = d#2049-4-18 AND x;
x := easter(2050) = d#2050-4-10 AND x;
x := easter(2051) = d#2051-4-2 AND x;
x := easter(2052) = d#2052-4-21 AND x;
x := easter(2053) = d#2053-4-6 AND x;
x := easter(2054) = d#2054-3-29 AND x;
x := easter(2055) = d#2055-4-18 AND x;
x := easter(2056) = d#2056-4-2 AND x;
x := easter(2057) = d#2057-4-22 AND x;
x := easter(2058) = d#2058-4-14 AND x;
x := easter(2059) = d#2059-3-30 AND x;
x := easter(2060) = d#2060-4-18 AND x;
x := easter(2061) = d#2061-4-10 AND x;
x := easter(2062) = d#2062-3-26 AND x;
x := easter(2063) = d#2063-4-15 AND x;
x := easter(2064) = d#2064-4-6 AND x;
x := easter(2065) = d#2065-3-29 AND x;
x := easter(2066) = d#2066-4-11 AND x;
x := easter(2067) = d#2067-4-3 AND x;
x := easter(2068) = d#2068-4-22 AND x;
x := easter(2069) = d#2069-4-14 AND x;
x := easter(2070) = d#2070-3-30 AND x;
x := easter(2071) = d#2071-4-19 AND x;
x := easter(2072) = d#2072-4-10 AND x;
x := easter(2073) = d#2073-3-26 AND x;
x := easter(2074) = d#2074-4-15 AND x;
x := easter(2075) = d#2075-4-7 AND x;
x := easter(2076) = d#2076-4-19 AND x;
x := easter(2077) = d#2077-4-11 AND x;
x := easter(2078) = d#2078-4-3 AND x;
x := easter(2079) = d#2079-4-23 AND x;
x := easter(2080) = d#2080-4-7 AND x;
x := easter(2081) = d#2081-3-30 AND x;
x := easter(2082) = d#2082-4-19 AND x;
x := easter(2083) = d#2083-4-4 AND x;
x := easter(2084) = d#2084-3-26 AND x;
x := easter(2085) = d#2085-4-15 AND x;
x := easter(2086) = d#2086-3-31 AND x;
x := easter(2087) = d#2087-4-20 AND x;
x := easter(2088) = d#2088-4-11 AND x;
x := easter(2089) = d#2089-4-3 AND x;
x := easter(2090) = d#2090-4-16 AND x;
x := easter(2091) = d#2091-4-8 AND x;
x := easter(2092) = d#2092-3-30 AND x;
x := easter(2093) = d#2093-4-12 AND x;
x := easter(2094) = d#2094-4-4 AND x;
x := easter(2095) = d#2095-4-24 AND x;
x := easter(2096) = d#2096-4-15 AND x;
x := easter(2097) = d#2097-3-31 AND x;
x := easter(2098) = d#2098-4-20 AND x;
x := easter(2099) = d#2099-4-12 AND x;
easter_test := X;

(* revision history
hm		26. mar. 2008		rev 1.0
	original release

*)
END_FUNCTION

(* POU Time&Date/LEAP_YEAR, ST *)
FUNCTION LEAP_YEAR : BOOL
VAR_INPUT
	yr : INT;
END_VAR
VAR
END_VAR

(*
version 1.1	2 oct 2006
programmer 	hugo
tested by		tobias


leap_year is true if the tested year is a leap year  
  
*)
leap_year := SHL(yr,14) = 0;

(* this code was used prior to rev 1.1

IF yr MOD 400 = 0 THEN leap_year := TRUE;
ELSIF yr MOD 100 = 0 THEN leap_year := FALSE;
ELSIF yr MOD 4 =0 THEN leap_year := TRUE;
ELSE leap_year := FALSE;
END_IF;

*)

(* change history

hm 	2.10.2006		rev 1.1
	the function now works for any year from 1970 up to 2100

hm	1. oct 2007		rev 1.2
	chaged code for higher performance
*)
END_FUNCTION

(* POU Time&Date/LOCAL_TIME, ST *)
FUNCTION LOCAL_TIME : DT
VAR_INPUT
	utc : DT;
	time_zone_offset : INT;
	dst_enable: BOOL;
END_VAR
VAR
	tx : TIME;
END_VAR

(*
version 1.4	8 dec 2007
programmer 	hugo
tested by		tobias

localtime calculates the local time according to DSTenable and time_zone_offset.
the dst input only tells the function the dst (daylight savings time) is enabled but the calculation for summertime on and off is done by the function itself.
this means the dst input only tells the function to switch summertime on and off automatically or not.
the function will switch to summertime automatically at the specified time end of march and back end of october.
the summertime calculation is done according to european standards.
the input is world time (UTC) and a given time_zone_offset for any time_zone.

*)
tx := DWORD_TO_TIME(INT_TO_DWORD(ABS(time_zone_offset))* 3600000);

IF DST(utc) AND dst_enable THEN
	IF time_zone_offset < 0 THEN local_time := utc - tx + T#1h; ELSE local_time := utc + tx + T#1h; END_IF;
ELSE
	IF time_zone_offset < 0 THEN local_time := utc - tx; ELSE local_time := utc + tx; END_IF;
END_IF;


(*

change history

2.10.2006 hm	rev 1.1
	corrected an error in the dst check for correct function

24. oct 2007	rev 1.2
	changed dst calculation because function dst was upgraded no error in DCF77 only a change in DST

12. nov 2007	rev 1.3
	changed time_zone_offset from time to integer to allow for negative offset time zones

8 dec 2007		rev 1.4
	corrected a problem with time_zone_offset
*)
END_FUNCTION

(* POU Time&Date/LTIME_TO_UTC, ST *)
FUNCTION LTIME_TO_UTC : DT
VAR_INPUT
	Ltime : DT;
	DST : BOOL;
	Time_Zone_Offset : INT;
END_VAR
VAR
	dst_offset : TIME := T#1h;
	tx: TIME;
END_VAR

(*
version 1.3	8 dec 2007
programmer 	hugo
tested by	tobias

LTIME_TO_UTC calculates UTC (World Time) from a local time LTIME. utc is calculated 
by subtracting Time_Zone_Offset from ltime and if dst it true subtracting an additional hour from ltime.

*)
(* convert integer time_zone_offset to hours *)
tx := DWORD_TO_TIME(INT_TO_DWORD(ABS(time_zone_offset))* 3600000);

IF DST THEN
	IF time_zone_offset < 0 THEN
		Ltime_to_UTC := Ltime + tx - dst_offset;
	ELSE
		Ltime_to_UTC := Ltime - tx - dst_offset;
	END_IF;
ELSE
	IF time_zone_offset < 0 THEN
		Ltime_to_UTC := Ltime + tx;
	ELSE
		Ltime_to_UTC := Ltime - tx;
	END_IF;
END_IF;



(* revision history
hm 5.7.2007		rev 1.0		
	original version

hm 5.11.2007	rev 1.1
	replaced literal constant with variable because of error in möller ecp4 compiler

hm	12.nov 2007	rev 1.2
	changed Type of time_zone_offset from time to int to allow for time zones with negative offset

hm	8. dec 2007	rev 1.3
	corrected a problem with time_zone_offset
*)
END_FUNCTION

(* POU Time&Date/LTIME, ST *)
FUNCTION_BLOCK LTIME
VAR_INPUT
	UTC : DT;
	dst_enable : BOOL;
	time_zone_offset : INT;
END_VAR
VAR_OUTPUT
	local_DT : DT;
	DST_on : BOOL;
	wday : INT;
END_VAR
VAR
	tx: TIME;
END_VAR

(*

version 1.6	8 dec 2007
programmer 	oscat
tested by		tobias

ltime is a real time clock that uses the system rtc as utc time and calculates and given time zone.
the utc time is supplied on the input UTC.
according to the input variable time_zone_offset when the input dst_enable is true,
the dst on and off times are calculated by a formula for any given year and the time is advanced and reset by one hour
at 02:00 and 03:00 for the last sunday of march and last sunday of october.
the code is high performance and the rtc counts every second.
if more then one time zone is needed by the systen the clock can be started many times by placing more then one function block.

execution time on wago 750-841 = 20 us 
 
*)
tx := DWORD_TO_TIME(INT_TO_DWORD(ABS(time_zone_offset))* 3600000);
DST_ON := DST(UTC) AND dst_enable;
IF DST_ON THEN
	IF time_zone_offset < 0 THEN local_DT := UTC - tx + t#1h; ELSE local_DT := UTC + tx + t#1h; END_IF;
ELSE
	IF time_zone_offset < 0 THEN local_DT := UTC - tx; ELSE local_DT := UTC + tx; END_IF;
END_IF;
wday := weekday(DT_TO_DATE(local_DT));


(* revision history

hm 2.10.2006	rev 1.1
	corrected an error where dst would be delayed by 0.1second

hm 17.1.2007	rev 1.2
	added utc input instead of internal sysrtcgettime because this would only work on wago.
	dst_enable would not be checked before dst would be enabled.

hm 18.3.2007	rev 1.3
	changed code, dst would not work during first cycle.

hm 24.10.2007	rev 1.4
	changed code because the execution every 100ms can cause major problems if the supplied time was not correct at start.
	use of new dst function

hm 12. nov 2007	rev 1.5
		changed Type of time_zone_offset from time to int to allow for time zones with negative offset

8 dec 2007		rev 1.6
	corrected a problem with time_zone_offset
*)
END_FUNCTION_BLOCK

(* POU Time&Date/PERIOD, ST *)
FUNCTION PERIOD : BOOL
VAR_INPUT
	d1 : DATE;
	dx : DATE;
	d2 : DATE;
END_VAR
VAR
	day1, day2, dayx : INT;
END_VAR

(*
version 1.3	22. mar. 2008
programmer 	hugo
tested by		tobias

PERIOD checks if a given date is between two dates (d1 and d2) d1 is the starting date and d2 the last date for the period.
the years of the dates are ignored, so the function period cheks for a time period within a year independet of the year.

*)
day1 := day_of_year(d1);
day2 := day_of_year(d2);
dayx := day_of_year(dx);
IF NOT leap_of_Date(dx) AND dayx > 58 THEN dayx := dayx + 1; END_IF;
IF NOT leap_of_Date(d1) AND day1 > 58 THEN day1 :=day1 + 1; END_IF;
IF NOT leap_of_Date(d2) AND day2 > 58 THEN day2 := day2 + 1; END_IF;

IF day2 < day1 THEN
	(* the period spans over the new year *)
	period := dayx <= day2 OR dayx >= day1;
ELSE
	period := dayx >= day1 AND dayx <= day2;
END_IF;

(* code before rev 1.2
yx := year(dx);
p1 := date_add(d1,0,0,0,yx - year(d1));
p2 := date_add(d2,0,0,0,yx - year(d2));

IF p2 >= p1 THEN
	period := dx <= p2  AND dx >= p1;
ELSE
	period := dx <= p2 OR dx >= p1;
END_IF;
*)


(* revision history

hm		19. sep 2007	rev 1.0
	original version

hm		20. sep 2007	rev 1.1
	corrected a problem with leap year

hm		4. jan 2008		rev 1.2
	changed code for better performance

hm		22. mar. 2008	rev 1.3
	function would deliver wrong results when d1, d2 or dx are a leap_year

*)
END_FUNCTION

(* POU XTEST/Testprojekt/TEST Routines/work_week_test, ST *)
FUNCTION work_week_test : BOOL
VAR_INPUT
END_VAR
VAR
	dx: DATE;
	y : ARRAY[0..30] OF INT := 1990,1991,1992,1993,1993,1994,1994,1995,1995,1996,1997,1998,1999,1999,2000,2000,2001,2002,2003,2004,2005,2005,2006,2006,2007,2008,2009,2010,2010,2011,2011;
	w : ARRAY[0..30] OF INT := 1,	1,	 1,   53,  1,   52,	 1,   52,  1,   1,   1,   1,   53,  1,   52,  1,   1,   1,   1,   1,   53,  1,   52,  1,   1,	1,   1,	  53,  1,   52,  1;
	d : ARRAY[0..30] OF INT := 7,	6,	 5,	  3,   10,  2,   9,   1,   8,   7,   5,   4,   3,   10,  2,   9,   7,   6,   5,   4,   2,   9,   1,   8,   7,	6,	 4,	  3,   10,  2,   9;
	i: INT;
	comp: INT;
	d1: DATE;
	day: INT;
	week: INT;
	yr: INT;
END_VAR
work_week_test := TRUE;
FOR i := 0 TO 30 DO
	day := d[i];
	week := w[i];
	yr := y[i];
	d1 := set_Date(yr,1,day);
	comp := work_week(d1);
	IF comp <> week THEN
		work_week_test := FALSE;
		dx := d1;
	END_IF;
	d1 := date_add(d1,-6,0,0,0);
	comp := work_week(d1);
	IF comp <> week THEN
		work_week_test := FALSE;
		dx := d1;
	END_IF;
END_FOR;


(* revision history
hm		26. mar. 2008		rev 1.0
	original release

*)
END_FUNCTION

(* POU Time&Date/WORK_WEEK, ST *)
FUNCTION WORK_WEEK : INT
VAR_INPUT
	idate : DATE;
END_VAR
VAR
	d1 : DATE;
	w1 : INT;
	ds: DWORD;
	yr: INT;
	w31: INT;
	w01: INT;
	wm: INT;
END_VAR

(*
version 1.3	16 mar 2008
programmer 	hugo
tested by		tobias

calculates the work week for a given date according to iso8601

*)
(* berechne den 1.1 des jahres von idate. *)
yr := year(idate);
d1 := year_begin(yr);
(* wochentag von d1 *)
w1 := weekday(d1);
(* offset des montags der eletzten KW des vorjahres *)
(* wenn der erste tag des jahres größer als donnerstag ist dann beginnt die letzte kw am montag davor *)
(* wenn der erste tag des jahres ein donnerstag oder kleiner ist beginnt die erste kw 2 montage davor *)
IF w1 < 5 THEN
	ds := DATE_TO_DWORD(d1) - INT_TO_DWORD(w1+6) * 86400;
ELSE
	ds := DATE_TO_DWORD(d1) - INT_TO_DWORD(w1-1) * 86400;
END_IF;

(* kalenderwoche des eingangsdatums *)
work_week := DWORD_TO_INT((DATE_TO_DWORD(idate) - ds) / 604800);

(* korrektur wenn work_week = 0 *)
IF work_week = 0 THEN
	(* work_week needs to be 53 when 1.jan of the year before is thursday or dec 31. is thursday. *)
	(* first and last weekday of a year is equal and one more day for a leap_year. *)
	IF w1 > 1 THEN w31 := w1 - 1; ELSE W31 := 7; END_IF;
	IF leap_year(yr - 1) THEN IF w31 > 1 THEN w01 := W31 - 1; ELSE w1 := 7; END_IF; END_IF;
	(* if first or last day of a year is a thursday, the year has 53 weeks *)
	IF w31 = 4 OR w01 = 4 THEN work_week := 53; ELSE work_week := 52; END_IF;
ELSE
	(* end of year calculation *)
	(* calculated the first and last weekday *)
	IF leap_year(yr) THEN
		IF w1 < 7 THEN w31 := w1 + 1; ELSE w31 := 1; END_IF;
	ELSE
		w31 := w1;
	END_IF;
	(* if first or last day is thursday then the year has 53 weeks otherwise only 52 *)
	IF w31 = 4 OR w1 = 4 THEN wm := 53; ELSE wm := 52; END_IF;
	IF work_week > wm THEN work_week := 1; END_IF;
END_IF;



(* old code before rev 1.2
w1 := weekday(set_Date(year(idate), 1,1));
IF w1 < 5 THEN
	work_week := (day_of_year(idate) + w1 + 5)/7;
ELSE
	work_week := (day_of_year(idate) + w1 - 2)/7;
END_IF
*)


(* revision history

hm 17.1.2007		rev 1.1
	deleted unused variable yday

hm	19. dec 2007	rev 1.2
	changed code for better performance
	changed code to comply with ISO8601

hm	16. mar 2008	rev 1.3
	added type conversions to avoid warnings under codesys 3.0
*)
END_FUNCTION

(* POU XTEST/Testprojekt/math_test, ST *)
FUNCTION_BLOCK math_test
VAR_INPUT
END_VAR
VAR_OUTPUT
	good : BOOL;

END_VAR
VAR CONSTANT
	N : INT := 6;	(* internal resolution in digits *)
END_VAR
VAR
	test: STRING;
	x : REAL;
	y : REAL;
	c : REAL;
	init : BOOL;
	rx : REAL;
END_VAR
IF NOT init THEN
	init := TRUE;
ELSIF NOT good THEN
	RETURN;
ELSE
	good := FALSE;
END_IF;

(* prepare random numbers *)
rx := RDM(rx);

(* test D_trunc *)
test := 'd_trunc';
IF D_TRUNC(0) <> 0 THEN RETURN; END_IF;
IF D_TRUNC(5) <> 5 THEN RETURN; END_IF;
IF D_TRUNC(0.0001) <> 0 THEN RETURN; END_IF;
IF D_TRUNC(0.5) <> 0 THEN RETURN; END_IF;
IF D_TRUNC(0.999) <> 0 THEN RETURN; END_IF;
IF D_TRUNC(-1.5) <> -1 THEN RETURN; END_IF;
IF D_TRUNC(-1.999) <> -1 THEN RETURN; END_IF;
IF D_TRUNC(-1.0001) <> -1 THEN RETURN; END_IF;
IF D_TRUNC(-5) <> -5 THEN RETURN; END_IF;

(* test cmp *)
test := 'cmp';
IF CMP(3.140,3.149,3) = FALSE THEN RETURN; END_IF;
IF CMP(4.2,4.0,2) = TRUE THEN RETURN; END_IF;
IF CMP(0.03140,0.03149,3) = FALSE THEN RETURN; END_IF;
IF CMP(0,0,1) = FALSE THEN RETURN; END_IF;
IF CMP(0.030,0.032,2) = TRUE THEN RETURN; END_IF;

(* check rdm number for range *)
test := 'rdm range';
x := rx;
IF rx < 0 OR rx >= 1 THEN RETURN; END_IF;

(* test acosh 1 <= X < +inv *)
test := 'acosh';
x := rx * 100 + 1;
y := ACOSH(x);
c := LN(SQRT(X*X - 1)+x);
IF NOT CMP(c,y,n) THEN RETURN; END_IF;
test := 'acosh(1)';
y := ACOSH(1);
C := 0;
IF NOT CMP(c,y,n) THEN RETURN; END_IF;

(* test asinh -inv < X < +inv *)
test := 'asinh';
x := (rx-0.5) * 100;
y := asinH(x);
c := LN(SQRT(X*X + 1)+x);
IF NOT CMP(c,y,n) THEN RETURN; END_IF;
test := 'asinh(0)';
y := ASINH(0);
C := 0;
IF NOT CMP(c,y,n) THEN RETURN; END_IF;

